KUKA KRL program: MyProgram_335().src

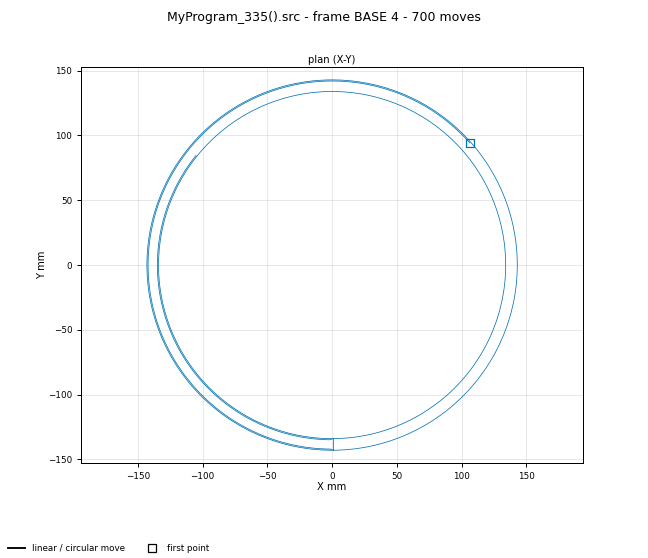
[picture p0: tool path of MyProgram_335().src in frame BASE 4, 700 of 700 moves have a stored position in this frame; points joined in program order, loops and branches not executed]
&ACCESS RVP
&REL 1
&PARAM TEMPLATE = C:\KRC\Roboter\Template\vorgabe
&PARAM EDITMASK = *
DEF MyProgram_335()
; ---- Setting reference (Base) ----
$BASE = BASE_DATA[4]

; --------------------------
; ---- Setting tool (TCP) ----
$TOOL = TOOL_DATA[3]
; --------------------------

$VEL.CP = VEL_APROX_PRINT
Startdeposition()
$VEL.CP = VEL_PRINT
LIN {X 106.2773,Y 94.2336,Z 189,A 42.7394,B 1.6929,C 0.0223,E1 1.815,E2 411.3828} C_DIS
LIN {X 103.2721,Y 97.5175,Z 189,A 44.3965,B 1.6929,C 0.0193,E1 1.8118,E2 409.7431} C_DIS
LIN {X 100.41,Y 100.4629,Z 189,A 45.7845,B 1.6929,C 0.0174,E1 1.8092,E2 408.3889} C_DIS
LIN {X 97.7243,Y 103.0771,Z 189,A 47.4179,B 1.693,C 0.0135,E1 1.8059,E2 406.7401} C_DIS
LIN {X 94.6798,Y 105.8799,Z 189,A 48.9807,B 1.693,C 0.0108,E1 1.8026,E2 405.1906} C_DIS
LIN {X 91.6362,Y 108.5256,Z 189,A 50.5192,B 1.693,C 0.0082,E1 1.7994,E2 403.6632} C_DIS
LIN {X 88.3912,Y 111.1836,Z 189,A 52.0959,B 1.693,C 0.0056,E1 1.796,E2 402.101} C_DIS
LIN {X 85.1125,Y 113.7136,Z 189,A 53.6495,B 1.693,C 0.0032,E1 1.7926,E2 400.562} C_DIS
LIN {X 81.9996,Y 115.978,Z 189,A 55.2099,B 1.693,C 0.0004,E1 1.789,E2 399.0007} C_DIS
LIN {X 78.1765,Y 118.5885,Z 189,A 56.9737,B 1.693,C -0.0023,E1 1.7849,E2 397.2499} C_DIS
LIN {X 74.3685,Y 121.013,Z 189,A 58.7195,B 1.693,C -0.0049,E1 1.7808,E2 395.5136} C_DIS
LIN {X 70.5126,Y 123.2996,Z 189,A 60.4494,B 1.693,C -0.0073,E1 1.7766,E2 393.7936} C_DIS
LIN {X 66.5595,Y 125.4767,Z 189,A 62.2164,B 1.693,C -0.0098,E1 1.7723,E2 392.0335} C_DIS
LIN {X 63.0559,Y 127.2723,Z 189,A 63.6578,B 1.693,C -0.0113,E1 1.7687,E2 390.6104} C_DIS
LIN {X 59.5637,Y 128.9434,Z 189,A 65.1264,B 1.693,C -0.013,E1 1.7651,E2 389.1536} C_DIS
LIN {X 56.8008,Y 130.185,Z 189,A 66.2211,B 1.693,C -0.014,E1 1.7623,E2 388.0748} C_DIS
LIN {X 54.0024,Y 131.372,Z 189,A 67.6332,B 1.693,C -0.0165,E1 1.7586,E2 386.64} C_DIS
LIN {X 50.101,Y 132.9068,Z 189,A 69.1211,B 1.693,C -0.0175,E1 1.7547,E2 385.1775} C_DIS
LIN {X 46.8537,Y 134.0862,Z 189,A 70.4786,B 1.693,C -0.019,E1 1.7512,E2 383.8248} C_DIS
LIN {X 40.2783,Y 136.206,Z 189,A 73.0708,B 1.693,C -0.021,E1 1.7443,E2 381.2572} C_DIS
LIN {X 36.9072,Y 137.1577,Z 189,A 74.5574,B 1.693,C -0.0227,E1 1.7403,E2 379.7619} C_DIS
LIN {X 33.8671,Y 137.9408,Z 189,A 75.7576,B 1.693,C -0.0236,E1 1.737,E2 378.5701} C_DIS
LIN {X 29.912,Y 138.8509,Z 189,A 77.2778,B 1.693,C -0.0244,E1 1.7329,E2 377.0648} C_DIS
LIN {X 27.0157,Y 139.4438,Z 189,A 78.5435,B 1.6929,C -0.0257,E1 1.7294,E2 375.7905} C_DIS
LIN {X 23.2743,Y 140.1165,Z 189,A 80.0251,B 1.6929,C -0.0266,E1 1.7253,E2 374.3156} C_DIS
LIN {X 19.566,Y 140.6833,Z 189,A 81.6158,B 1.6929,C -0.0279,E1 1.7209,E2 372.7159} C_DIS
LIN {X 15.4525,Y 141.1936,Z 189,A 83.1691,B 1.6929,C -0.0283,E1 1.7166,E2 371.1777} C_DIS
LIN {X 12.1084,Y 141.5195,Z 189,A 84.3357,B 1.6929,C -0.0283,E1 1.7134,E2 370.0346} C_DIS
LIN {X 9.4248,Y 141.7252,Z 189,A 85.5879,B 1.6929,C -0.0294,E1 1.7099,E2 368.7625} C_DIS
LIN {X 6.1391,Y 141.9051,Z 189,A 86.9513,B 1.6929,C -0.03,E1 1.706,E2 367.3953} C_DIS
LIN {X 1.6359,Y 142.029,Z 189,A 88.7776,B 1.6929,C -0.0306,E1 1.7009,E2 365.5686} C_DIS
LIN {X -2.4489,Y 142.0155,Z 189,A 90.3695,B 1.6929,C -0.0308,E1 1.6965,E2 363.9841} C_DIS
LIN {X -6.6903,Y 141.8796,Z 189,A 92.0648,B 1.6929,C -0.031,E1 1.6917,E2 362.2916} C_DIS
LIN {X -10.4141,Y 141.6542,Z 189,A 93.5286,B 1.6929,C -0.031,E1 1.6876,E2 360.8335} C_DIS
LIN {X -14.6574,Y 141.2792,Z 189,A 95.349,B 1.6928,C -0.0312,E1 1.6825,E2 359.0014} C_DIS
LIN {X -19.0699,Y 140.7518,Z 189,A 97.1416,B 1.6928,C -0.0311,E1 1.6775,E2 357.2096} C_DIS
LIN {X -22.6456,Y 140.2214,Z 189,A 98.4481,B 1.6928,C -0.0303,E1 1.674,E2 355.9224} C_DIS
LIN {X -26.2848,Y 139.5836,Z 189,A 99.9509,B 1.6928,C -0.0299,E1 1.6698,E2 354.4187} C_DIS
LIN {X -30.2845,Y 138.7705,Z 189,A 101.8492,B 1.6928,C -0.0302,E1 1.6645,E2 352.4905} C_DIS
LIN {X -34.665,Y 137.7415,Z 189,A 103.4007,B 1.6928,C -0.0286,E1 1.6604,E2 350.9722} C_DIS
LIN {X -38.3306,Y 136.7664,Z 189,A 105.04,B 1.6928,C -0.0282,E1 1.6559,E2 349.3203} C_DIS
LIN {X -41.5195,Y 135.8322,Z 189,A 106.3705,B 1.6928,C -0.0274,E1 1.6523,E2 347.9917} C_DIS
LIN {X -44.6408,Y 134.8389,Z 189,A 107.699,B 1.6928,C -0.0266,E1 1.6488,E2 346.6631} C_DIS
LIN {X -47.2057,Y 133.9641,Z 189,A 109.0092,B 1.6928,C -0.0264,E1 1.6453,E2 345.3271} C_DIS
LIN {X -51.3738,Y 132.4197,Z 189,A 110.6484,B 1.6929,C -0.0247,E1 1.641,E2 343.7076} C_DIS
LIN {X -53.9048,Y 131.4126,Z 189,A 111.9788,B 1.6929,C -0.0244,E1 1.6375,E2 342.3496} C_DIS
LIN {X -57.1041,Y 130.0538,Z 189,A 113.2798,B 1.6929,C -0.0228,E1 1.6342,E2 341.0619} C_DIS
LIN {X -60.454,Y 128.5312,Z 189,A 115.0186,B 1.6929,C -0.022,E1 1.6297,E2 339.2927} C_DIS
LIN {X -64.3455,Y 126.6249,Z 189,A 116.6404,B 1.6929,C -0.0199,E1 1.6257,E2 337.6873} C_DIS
LIN {X -67.2006,Y 125.1355,Z 189,A 118.1653,B 1.6929,C -0.019,E1 1.6218,E2 336.1356} C_DIS
LIN {X -71.656,Y 122.639,Z 189,A 120.235,B 1.693,C -0.0166,E1 1.6168,E2 334.066} C_DIS
LIN {X -75.5784,Y 120.2613,Z 189,A 122.1545,B 1.693,C -0.0143,E1 1.6122,E2 332.1392} C_DIS
LIN {X -79.4708,Y 117.7252,Z 189,A 124.0179,B 1.693,C -0.0118,E1 1.6078,E2 330.2783} C_DIS
LIN {X -83.1126,Y 115.1833,Z 189,A 125.9602,B 1.693,C -0.0095,E1 1.6034,E2 328.3184} C_DIS
LIN {X -86.7314,Y 112.4837,Z 189,A 127.8838,B 1.693,C -0.0069,E1 1.599,E2 326.3833} C_DIS
LIN {X -90.284,Y 109.6528,Z 189,A 129.7857,B 1.693,C -0.0041,E1 1.5949,E2 324.4741} C_DIS
LIN {X -93.551,Y 106.8787,Z 189,A 131.6035,B 1.693,C -0.0013,E1 1.591,E2 322.6463} C_DIS
LIN {X -96.9568,Y 103.799,Z 189,A 133.5203,B 1.693,C 0.0018,E1 1.5871,E2 320.7227} C_DIS
LIN {X -100.085,Y 100.7858,Z 189,A 135.4048,B 1.693,C 0.0048,E1 1.5833,E2 318.823} C_DIS
LIN {X -103.2004,Y 97.5936,Z 189,A 137.3305,B 1.693,C 0.008,E1 1.5795,E2 316.8826} C_DIS
LIN {X -106.2595,Y 94.2537,Z 189,A 139.2838,B 1.693,C 0.0114,E1 1.5758,E2 314.9147} C_DIS
LIN {X -109.2471,Y 90.774,Z 189,A 141.2114,B 1.693,C 0.0151,E1 1.5723,E2 312.9787} C_DIS
LIN {X -111.9901,Y 87.3683,Z 189,A 142.9572,B 1.693,C 0.0188,E1 1.5693,E2 311.2364} C_DIS
LIN {X -114.18,Y 84.4857,Z 189,A 144.7828,B 1.693,C 0.0214,E1 1.5661,E2 309.3657} C_DIS
LIN {X -117.2007,Y 80.2423,Z 189,A 146.9388,B 1.6929,C 0.026,E1 1.5627,E2 307.2043} C_DIS
LIN {X -119.775,Y 76.3468,Z 189,A 148.9107,B 1.6929,C 0.0302,E1 1.5597,E2 305.2224} C_DIS
LIN {X -122.0067,Y 72.7266,Z 189,A 150.7317,B 1.6927,C 0.0341,E1 1.557,E2 303.3893} C_DIS
LIN {X -124.3948,Y 68.5625,Z 189,A 152.8841,B 1.6927,C 0.0384,E1 1.554,E2 301.2106} C_DIS
LIN {X -126.4099,Y 64.7679,Z 189,A 154.6626,B 1.6925,C 0.0426,E1 1.5517,E2 299.4275} C_DIS
LIN {X -129.3506,Y 58.6788,Z 189,A 157.6639,B 1.6924,C 0.0491,E1 1.5481,E2 296.3931} C_DIS
LIN {X -131.2019,Y 54.4098,Z 189,A 159.744,B 1.6922,C 0.0537,E1 1.5458,E2 294.2881} C_DIS
LIN {X -132.6655,Y 50.7415,Z 189,A 161.5557,B 1.6922,C 0.0576,E1 1.5439,E2 292.4493} C_DIS
LIN {X -133.971,Y 47.1847,Z 189,A 162.9511,B 1.692,C 0.0617,E1 1.5426,E2 291.0722} C_DIS
LIN {X -135.1927,Y 43.5582,Z 189,A 164.6541,B 1.6918,C 0.0656,E1 1.5411,E2 289.3496} C_DIS
LIN {X -136.1268,Y 40.5488,Z 189,A 166.2155,B 1.6917,C 0.0688,E1 1.5398,E2 287.7514} C_DIS
LIN {X -138.2076,Y 32.7602,Z 189,A 169.5503,B 1.6913,C 0.0775,E1 1.5375,E2 284.408} C_DIS
LIN {X -139.5086,Y 26.6769,Z 189,A 172.3268,B 1.691,C 0.0842,E1 1.5359,E2 281.5983} C_DIS
LIN {X -140.4655,Y 21.0763,Z 189,A 174.9757,B 1.6907,C 0.0902,E1 1.5346,E2 278.9039} C_DIS
LIN {X -141.0217,Y 16.9484,Z 189,A 176.6676,B 1.6904,C 0.0949,E1 1.534,E2 277.2115} C_DIS
LIN {X -141.332,Y 14.1401,Z 189,A 177.8354,B 1.6902,C 0.098,E1 1.5337,E2 276.0408} C_DIS
LIN {X -141.6373,Y 10.6462,Z 189,A 179.4383,B 1.69,C 0.1018,E1 1.5333,E2 274.4138} C_DIS
LIN {X -141.8039,Y 8.1466,Z 189,A -179.2535,B 1.6899,C 0.1044,E1 1.5331,E2 273.0667} C_DIS
LIN {X -141.9587,Y 4.7647,Z 189,A -177.7459,B 1.6896,C 0.1081,E1 1.533,E2 271.5411} C_DIS
LIN {X -142.0388,Y -0.2591,Z 189,A -175.4645,B 1.6893,C 0.1136,E1 1.533,E2 269.2268} C_DIS
LIN {X -141.9528,Y -4.9149,Z 189,A -173.7364,B 1.6889,C 0.119,E1 1.533,E2 267.5199} C_DIS
LIN {X -141.8556,Y -7.1668,Z 189,A -172.5939,B 1.6887,C 0.1213,E1 1.5332,E2 266.3465} C_DIS
LIN {X -141.4766,Y -12.6168,Z 189,A -170.148,B 1.6883,C 0.1273,E1 1.5337,E2 263.8692} C_DIS
LIN {X -141.0326,Y -16.8571,Z 189,A -168.4784,B 1.6879,C 0.1321,E1 1.5342,E2 262.2073} C_DIS
LIN {X -140.629,Y -19.9456,Z 189,A -166.1435,B 1.6877,C 0.1346,E1 1.5353,E2 259.7262} C_DIS
LIN {X -139.6388,Y -25.996,Z 189,A -163.7081,B 1.6872,C 0.1414,E1 1.5365,E2 257.2973} C_DIS
LIN {X -138.6976,Y -30.6224,Z 189,A -162.0866,B 1.6867,C 0.1469,E1 1.5374,E2 255.7156} C_DIS
LIN {X -137.8516,Y -34.231,Z 189,A -160.4161,B 1.6864,C 0.1507,E1 1.5385,E2 254.0218} C_DIS
LIN {X -136.7518,Y -38.3827,Z 189,A -158.7867,B 1.6859,C 0.1555,E1 1.5397,E2 252.4073} C_DIS
LIN {X -135.9501,Y -41.1344,Z 189,A -157.4275,B 1.6857,C 0.1583,E1 1.5408,E2 251.0207} C_DIS
LIN {X -135.008,Y -44.133,Z 189,A -155.8637,B 1.6854,C 0.1613,E1 1.5422,E2 249.4167} C_DIS
LIN {X -133.8121,Y -47.6331,Z 189,A -154.5652,B 1.685,C 0.1654,E1 1.5434,E2 248.1456} C_DIS
LIN {X -132.7591,Y -50.4955,Z 189,A -152.9409,B 1.6847,C 0.1682,E1 1.545,E2 246.4674} C_DIS
LIN {X -131.2624,Y -54.2648,Z 189,A -151.4833,B 1.6843,C 0.1725,E1 1.5465,E2 245.035} C_DIS
LIN {X -128.9947,Y -59.4527,Z 189,A -148.7099,B 1.6837,C 0.1776,E1 1.5497,E2 242.1946} C_DIS
LIN {X -126.7671,Y -64.0663,Z 189,A -146.6066,B 1.6832,C 0.1826,E1 1.5523,E2 240.0869} C_DIS
LIN {X -125.0385,Y -67.3811,Z 189,A -144.9402,B 1.6828,C 0.186,E1 1.5546,E2 238.399} C_DIS
LIN {X -122.8547,Y -71.2849,Z 189,A -143.0116,B 1.6824,C 0.1901,E1 1.5572,E2 236.4535} C_DIS
LIN {X -121.0931,Y -74.2378,Z 189,A -141.2058,B 1.6821,C 0.1926,E1 1.56,E2 234.5893} C_DIS
LIN {X -119.1112,Y -77.3777,Z 189,A -140.0244,B 1.6816,C 0.1965,E1 1.5617,E2 233.4528} C_DIS
LIN {X -116.9843,Y -80.5575,Z 189,A -138.2365,B 1.6813,C 0.1995,E1 1.5645,E2 231.6308} C_DIS
LIN {X -115.1472,Y -83.1624,Z 189,A -136.5306,B 1.681,C 0.2016,E1 1.5675,E2 229.8659} C_DIS
LIN {X -112.8126,Y -86.3024,Z 189,A -135.1781,B 1.6806,C 0.2053,E1 1.5697,E2 228.5457} C_DIS
LIN {X -110.1042,Y -89.7324,Z 189,A -133.3246,B 1.6802,C 0.2088,E1 1.5729,E2 226.6797} C_DIS
LIN {X -108.1098,Y -92.1254,Z 189,A -131.8953,B 1.6799,C 0.211,E1 1.5756,E2 225.2261} C_DIS
LIN {X -104.9235,Y -95.7393,Z 189,A -129.8541,B 1.6794,C 0.2145,E1 1.5794,E2 223.1713} C_DIS
LIN {X -101.7136,Y -99.143,Z 189,A -127.698,B 1.6791,C 0.2175,E1 1.5837,E2 220.9771} C_DIS
LIN {X -98.0261,Y -102.7896,Z 189,A -125.6758,B 1.6786,C 0.2214,E1 1.5877,E2 218.965} C_DIS
LIN {X -94.5718,Y -105.9766,Z 189,A -123.6873,B 1.6781,C 0.2244,E1 1.5919,E2 216.9634} C_DIS
LIN {X -91.0557,Y -109.0126,Z 189,A -121.6766,B 1.6778,C 0.2271,E1 1.5962,E2 214.9332} C_DIS
LIN {X -87.3782,Y -111.9823,Z 189,A -119.7857,B 1.6774,C 0.2301,E1 1.6003,E2 213.0446} C_DIS
LIN {X -83.6065,Y -114.8253,Z 189,A -117.6892,B 1.6771,C 0.2325,E1 1.6051,E2 210.9206} C_DIS
LIN {X -79.8824,Y -117.4466,Z 189,A -115.7606,B 1.6767,C 0.2348,E1 1.6096,E2 208.9788} C_DIS
LIN {X -75.983,Y -120.0059,Z 189,A -113.8584,B 1.6764,C 0.2372,E1 1.6141,E2 207.0734} C_DIS
LIN {X -72.2327,Y -122.3002,Z 189,A -111.9585,B 1.6761,C 0.239,E1 1.6187,E2 205.1552} C_DIS
LIN {X -68.162,Y -124.6145,Z 189,A -110.0444,B 1.6758,C 0.241,E1 1.6234,E2 203.2372} C_DIS
LIN {X -64.7484,Y -126.4198,Z 189,A -108.5031,B 1.6756,C 0.2427,E1 1.6272,E2 201.698} C_DIS
LIN {X -61.576,Y -127.9952,Z 189,A -107.1255,B 1.6754,C 0.2443,E1 1.6307,E2 200.3275} C_DIS
LIN {X -58.3162,Y -129.5128,Z 189,A -105.7448,B 1.6751,C 0.2459,E1 1.6342,E2 198.9566} C_DIS
LIN {X -55.7418,Y -130.6428,Z 189,A -104.2642,B 1.6751,C 0.2457,E1 1.6381,E2 197.4258} C_DIS
LIN {X -51.8273,Y -132.2434,Z 189,A -102.6432,B 1.6749,C 0.2473,E1 1.6423,E2 195.8167} C_DIS
LIN {X -48.4711,Y -133.5099,Z 189,A -101.2597,B 1.6747,C 0.2486,E1 1.6459,E2 194.442} C_DIS
LIN {X -43.7182,Y -135.1416,Z 189,A -98.9872,B 1.6747,C 0.249,E1 1.652,E2 192.1334} C_DIS
LIN {X -39.1432,Y -136.5384,Z 189,A -97.0299,B 1.6745,C 0.2499,E1 1.6573,E2 190.1717} C_DIS
LIN {X -34.3439,Y -137.8229,Z 189,A -94.9798,B 1.6745,C 0.2506,E1 1.6629,E2 188.1142} C_DIS
LIN {X -30.6716,Y -138.6869,Z 189,A -93.6287,B 1.6743,C 0.2518,E1 1.6665,E2 186.7874} C_DIS
LIN {X -27.0587,Y -139.4356,Z 189,A -91.9873,B 1.6743,C 0.2516,E1 1.6711,E2 185.1231} C_DIS
LIN {X -23.8319,Y -140.0235,Z 189,A -90.8191,B 1.6742,C 0.2525,E1 1.6743,E2 183.9769} C_DIS
LIN {X -20.9337,Y -140.4876,Z 189,A -89.3995,B 1.6742,C 0.2517,E1 1.6783,E2 182.5227} C_DIS
LIN {X -16.9659,Y -141.0196,Z 189,A -88.0583,B 1.6741,C 0.253,E1 1.6819,E2 181.2205} C_DIS
LIN {X -14.208,Y -141.3255,Z 189,A -86.8707,B 1.6741,C 0.2527,E1 1.6853,E2 180.0226} C_DIS
LIN {X -10.3399,Y -141.6596,Z 189,A -85.1907,B 1.6742,C 0.2521,E1 1.69,E2 178.3253} C_DIS
LIN {X -5.7286,Y -141.9211,Z 189,A -83.3211,B 1.6742,C 0.2519,E1 1.6953,E2 176.4539} C_DIS
LIN {X -1.1428,Y -142.0324,Z 189,A -81.5425,B 1.6742,C 0.2518,E1 1.7002,E2 174.6848} C_DIS
LIN {X -1.1428,Y -142.0324,Z 189,A -81.5425,B 1.6742,C 0.2518,E1 1.7002,E2 174.6848} C_DIS
Enddeposition()
LIN {X 1.0097,Y -142.9296,Z 189,A -80.9147,B 1.6738,C 0.2534,E1 1.7016,E2 174.1194} C_DIS
Startdeposition()
$VEL.CP = VEL_PRINT
LIN {X -1.408,Y -142.9302,Z 189,A -82.2099,B 1.6736,C 0.2552,E1 1.6979,E2 175.4628} C_DIS
LIN {X -5.2622,Y -142.8391,Z 189,A -83.6981,B 1.6736,C 0.2552,E1 1.6937,E2 176.9434} C_DIS
LIN {X -8.4198,Y -142.6879,Z 189,A -85.1105,B 1.6734,C 0.256,E1 1.6897,E2 178.3774} C_DIS
LIN {X -12.2561,Y -142.4094,Z 189,A -86.5262,B 1.6735,C 0.2555,E1 1.6858,E2 179.7755} C_DIS
LIN {X -15.4038,Y -142.1032,Z 189,A -87.8442,B 1.6735,C 0.2557,E1 1.6821,E2 181.1013} C_DIS
LIN {X -19.2397,Y -141.6364,Z 189,A -89.3872,B 1.6735,C 0.2557,E1 1.6778,E2 182.6442} C_DIS
LIN {X -22.7055,Y -141.123,Z 189,A -90.8211,B 1.6735,C 0.2555,E1 1.6738,E2 184.083} C_DIS
LIN {X -25.7283,Y -140.602,Z 189,A -92.0459,B 1.6735,C 0.2552,E1 1.6704,E2 185.3074} C_DIS
LIN {X -29.4561,Y -139.8692,Z 189,A -93.6335,B 1.6735,C 0.255,E1 1.666,E2 186.905} C_DIS
LIN {X -33.0187,Y -139.0702,Z 189,A -95.0391,B 1.6737,C 0.2543,E1 1.6622,E2 188.3027} C_DIS
LIN {X -36.4297,Y -138.2157,Z 189,A -96.3842,B 1.6738,C 0.2535,E1 1.6586,E2 189.6389} C_DIS
LIN {X -39.7974,Y -137.2837,Z 189,A -97.8075,B 1.6739,C 0.2529,E1 1.6547,E2 191.066} C_DIS
LIN {X -42.824,Y -136.3712,Z 189,A -99.198,B 1.6739,C 0.2526,E1 1.6509,E2 192.4747} C_DIS
LIN {X -46.4642,Y -135.1729,Z 189,A -100.6617,B 1.6741,C 0.2514,E1 1.6471,E2 193.9283} C_DIS
LIN {X -49.0106,Y -134.2712,Z 189,A -102.0278,B 1.6741,C 0.2516,E1 1.6434,E2 195.3356} C_DIS
LIN {X -53.0801,Y -132.7144,Z 189,A -103.5446,B 1.6744,C 0.2495,E1 1.6395,E2 196.8196} C_DIS
LIN {X -56.0011,Y -131.5103,Z 189,A -104.9545,B 1.6745,C 0.2489,E1 1.6358,E2 198.2506} C_DIS
LIN {X -58.7218,Y -130.3164,Z 189,A -106.1866,B 1.6746,C 0.248,E1 1.6326,E2 199.4888} C_DIS
LIN {X -61.8977,Y -128.838,Z 189,A -107.6334,B 1.6748,C 0.2468,E1 1.6289,E2 200.942} C_DIS
LIN {X -65.0427,Y -127.279,Z 189,A -109.0825,B 1.675,C 0.2455,E1 1.6253,E2 202.3974} C_DIS
LIN {X -68.3071,Y -125.5595,Z 189,A -110.7111,B 1.6752,C 0.2443,E1 1.6212,E2 204.0477} C_DIS
LIN {X -71.9805,Y -123.491,Z 189,A -112.3949,B 1.6755,C 0.2423,E1 1.6171,E2 205.7309} C_DIS
LIN {X -75.5848,Y -121.3177,Z 189,A -114.1419,B 1.6757,C 0.2404,E1 1.6129,E2 207.4866} C_DIS
LIN {X -79.2667,Y -118.9447,Z 189,A -115.9737,B 1.676,C 0.2383,E1 1.6086,E2 209.3295} C_DIS
LIN {X -82.4457,Y -116.7637,Z 189,A -117.6742,B 1.6763,C 0.2366,E1 1.6046,E2 211.0522} C_DIS
LIN {X -85.9738,Y -114.1909,Z 189,A -119.4814,B 1.6766,C 0.2341,E1 1.6006,E2 212.8677} C_DIS
LIN {X -89.4478,Y -111.4911,Z 189,A -121.3704,B 1.677,C 0.2317,E1 1.5964,E2 214.7746} C_DIS
LIN {X -92.704,Y -108.7981,Z 189,A -123.1445,B 1.6773,C 0.2292,E1 1.5925,E2 216.56} C_DIS
LIN {X -96.115,Y -105.7967,Z 189,A -125.0599,B 1.6777,C 0.2263,E1 1.5885,E2 218.4887} C_DIS
LIN {X -99.3067,Y -102.8068,Z 189,A -126.8794,B 1.6781,C 0.2233,E1 1.5848,E2 220.3175} C_DIS
LIN {X -102.2872,Y -99.8423,Z 189,A -128.5767,B 1.6785,C 0.2203,E1 1.5815,E2 222.0164} C_DIS
LIN {X -105.2002,Y -96.7675,Z 189,A -130.4002,B 1.6789,C 0.2173,E1 1.5779,E2 223.8574} C_DIS
LIN {X -108.0446,Y -93.5818,Z 189,A -132.2121,B 1.6793,C 0.2142,E1 1.5746,E2 225.6833} C_DIS
LIN {X -110.4898,Y -90.6814,Z 189,A -133.9376,B 1.6796,C 0.2115,E1 1.5714,E2 227.4374} C_DIS
LIN {X -113.2109,Y -87.261,Z 189,A -135.7018,B 1.6801,C 0.2078,E1 1.5684,E2 229.203} C_DIS
LIN {X -115.7265,Y -83.8952,Z 189,A -137.5131,B 1.6805,C 0.2045,E1 1.5653,E2 231.0318} C_DIS
LIN {X -118.2614,Y -80.2827,Z 189,A -139.3933,B 1.681,C 0.2008,E1 1.5623,E2 232.9272} C_DIS
LIN {X -120.365,Y -77.0927,Z 189,A -141.1327,B 1.6813,C 0.1976,E1 1.5596,E2 234.6953} C_DIS
LIN {X -122.6017,Y -73.4845,Z 189,A -142.9789,B 1.6818,C 0.1939,E1 1.5569,E2 236.5612} C_DIS
LIN {X -124.8787,Y -69.5448,Z 189,A -144.9149,B 1.6822,C 0.1898,E1 1.5542,E2 238.5123} C_DIS
LIN {X -126.7901,Y -65.9924,Z 189,A -146.5547,B 1.6827,C 0.186,E1 1.5521,E2 240.1547} C_DIS
LIN {X -128.3777,Y -62.8474,Z 189,A -148.0738,B 1.683,C 0.1827,E1 1.5502,E2 241.6881} C_DIS
LIN {X -129.8804,Y -59.6797,Z 189,A -149.5912,B 1.6834,C 0.1793,E1 1.5483,E2 243.2205} C_DIS
LIN {X -131.3588,Y -56.3515,Z 189,A -151.1443,B 1.6838,C 0.1758,E1 1.5466,E2 244.786} C_DIS
LIN {X -132.7165,Y -53.0751,Z 189,A -152.664,B 1.6841,C 0.1723,E1 1.545,E2 246.3187} C_DIS
LIN {X -133.8564,Y -50.1293,Z 189,A -154.1378,B 1.6844,C 0.1693,E1 1.5435,E2 247.8206} C_DIS
LIN {X -135.1558,Y -46.5134,Z 189,A -155.7021,B 1.6848,C 0.1653,E1 1.542,E2 249.3876} C_DIS
LIN {X -136.158,Y -43.4913,Z 189,A -157.1951,B 1.6851,C 0.1622,E1 1.5407,E2 250.9097} C_DIS
LIN {X -137.2796,Y -39.8117,Z 189,A -158.7686,B 1.6855,C 0.1581,E1 1.5395,E2 252.4869} C_DIS
LIN {X -138.1263,Y -36.7647,Z 189,A -160.1953,B 1.6858,C 0.1549,E1 1.5384,E2 253.9348} C_DIS
LIN {X -138.9874,Y -33.3623,Z 189,A -161.7271,B 1.6861,C 0.1512,E1 1.5374,E2 255.4829} C_DIS
LIN {X -139.7645,Y -29.941,Z 189,A -163.2595,B 1.6865,C 0.1475,E1 1.5364,E2 257.0318} C_DIS
LIN {X -140.5199,Y -26.1755,Z 189,A -164.912,B 1.6868,C 0.1434,E1 1.5355,E2 258.6989} C_DIS
LIN {X -141.0622,Y -23.0699,Z 189,A -166.3064,B 1.6871,C 0.1401,E1 1.5349,E2 260.1104} C_DIS
LIN {X -141.5904,Y -19.5744,Z 189,A -167.8479,B 1.6874,C 0.1363,E1 1.5342,E2 261.668} C_DIS
LIN {X -142.0642,Y -15.7664,Z 189,A -169.5501,B 1.6877,C 0.1321,E1 1.5337,E2 263.3914} C_DIS
LIN {X -142.4066,Y -12.2889,Z 189,A -170.9826,B 1.688,C 0.1282,E1 1.5333,E2 264.8274} C_DIS
LIN {X -142.6438,Y -9.1356,Z 189,A -172.5371,B 1.6883,C 0.1249,E1 1.533,E2 266.4197} C_DIS
LIN {X -142.8393,Y -5.2579,Z 189,A -174.0995,B 1.6886,C 0.1206,E1 1.5328,E2 267.982} C_DIS
LIN {X -142.9205,Y -2.1023,Z 189,A -175.517,B 1.6888,C 0.1172,E1 1.5328,E2 269.4191} C_DIS
LIN {X -142.9314,Y 1.2571,Z 189,A -177.1181,B 1.6891,C 0.1136,E1 1.5328,E2 271.0533} C_DIS
LIN {X -142.8394,Y 5.2564,Z 189,A -178.6726,B 1.6894,C 0.1091,E1 1.5328,E2 272.6004} C_DIS
LIN {X -142.6874,Y 8.4286,Z 189,A 179.7693,B 1.6896,C 0.1057,E1 1.5331,E2 274.1955} C_DIS
LIN {X -142.4177,Y 12.1579,Z 189,A 178.2546,B 1.6899,C 0.1016,E1 1.5334,E2 275.7114} C_DIS
LIN {X -142.1033,Y 15.4032,Z 189,A 176.7863,B 1.6901,C 0.098,E1 1.5339,E2 277.2001} C_DIS
LIN {X -141.6393,Y 19.2174,Z 189,A 175.1147,B 1.6903,C 0.0939,E1 1.5345,E2 278.8881} C_DIS
LIN {X -141.1264,Y 22.6839,Z 189,A 173.5843,B 1.6905,C 0.0901,E1 1.5351,E2 280.4341} C_DIS
LIN {X -140.6101,Y 25.6829,Z 189,A 172.2359,B 1.6907,C 0.0868,E1 1.5358,E2 281.7985} C_DIS
LIN {X -139.8447,Y 29.5695,Z 189,A 170.5028,B 1.6909,C 0.0826,E1 1.5367,E2 283.5496} C_DIS
LIN {X -139.082,Y 32.97,Z 189,A 168.9809,B 1.6911,C 0.0789,E1 1.5377,E2 285.0868} C_DIS
LIN {X -138.1442,Y 36.6977,Z 189,A 167.2273,B 1.6912,C 0.0749,E1 1.539,E2 286.867} C_DIS
LIN {X -136.8823,Y 41.1612,Z 189,A 165.2802,B 1.6915,C 0.07,E1 1.5405,E2 288.8243} C_DIS
LIN {X -135.7167,Y 44.8505,Z 189,A 163.5964,B 1.6916,C 0.066,E1 1.5419,E2 290.5241} C_DIS
LIN {X -134.6949,Y 47.8354,Z 189,A 162.2243,B 1.6917,C 0.0628,E1 1.5432,E2 291.9093} C_DIS
LIN {X -133.455,Y 51.1924,Z 189,A 160.5899,B 1.6919,C 0.0592,E1 1.5448,E2 293.5684} C_DIS
LIN {X -132.1903,Y 54.3763,Z 189,A 159.1817,B 1.6919,C 0.0557,E1 1.5463,E2 294.9801} C_DIS
LIN {X -130.8136,Y 57.6102,Z 189,A 157.6716,B 1.6921,C 0.0523,E1 1.548,E2 296.5022} C_DIS
LIN {X -129.5944,Y 60.2982,Z 189,A 156.3682,B 1.6921,C 0.0494,E1 1.5496,E2 297.8201} C_DIS
LIN {X -127.7947,Y 64.0292,Z 189,A 154.5685,B 1.6923,C 0.0455,E1 1.5518,E2 299.6366} C_DIS
LIN {X -126.1391,Y 67.2322,Z 189,A 153.0106,B 1.6923,C 0.0421,E1 1.5538,E2 301.2078} C_DIS
LIN {X -124.3581,Y 70.4717,Z 189,A 151.4211,B 1.6925,C 0.0387,E1 1.556,E2 302.8098} C_DIS
LIN {X -122.5083,Y 73.6403,Z 189,A 149.7209,B 1.6925,C 0.0355,E1 1.5585,E2 304.538} C_DIS
LIN {X -120.2912,Y 77.2081,Z 189,A 147.8888,B 1.6926,C 0.0318,E1 1.5612,E2 306.3876} C_DIS
LIN {X -117.7768,Y 80.9919,Z 189,A 145.9368,B 1.6926,C 0.0278,E1 1.5643,E2 308.3548} C_DIS
LIN {X -114.9265,Y 84.989,Z 189,A 143.8604,B 1.6927,C 0.0237,E1 1.5677,E2 310.4434} C_DIS
LIN {X -112.143,Y 88.6294,Z 189,A 141.9924,B 1.6927,C 0.0198,E1 1.571,E2 312.3141} C_DIS
LIN {X -109.8275,Y 91.4829,Z 189,A 140.2818,B 1.6928,C 0.0171,E1 1.5741,E2 314.0533} C_DIS
LIN {X -106.6192,Y 95.202,Z 189,A 138.2635,B 1.6928,C 0.0133,E1 1.5778,E2 316.0764} C_DIS
LIN {X -103.5205,Y 98.5628,Z 189,A 136.3937,B 1.6928,C 0.0098,E1 1.5814,E2 317.9495} C_DIS
LIN {X -101.0738,Y 101.0709,Z 189,A 134.7774,B 1.6928,C 0.0075,E1 1.5846,E2 319.5912} C_DIS
LIN {X -97.9296,Y 104.1195,Z 189,A 132.9049,B 1.6928,C 0.0046,E1 1.5884,E2 321.477} C_DIS
LIN {X -94.5507,Y 107.1971,Z 189,A 130.9743,B 1.6928,C 0.0016,E1 1.5925,E2 323.4185} C_DIS
LIN {X -90.8118,Y 110.3832,Z 189,A 128.9328,B 1.6928,C -0.0015,E1 1.5969,E2 325.4676} C_DIS
LIN {X -87.2518,Y 113.218,Z 189,A 127.0909,B 1.6928,C -0.0044,E1 1.6009,E2 327.3105} C_DIS
LIN {X -83.8809,Y 115.7369,Z 189,A 125.3172,B 1.6928,C -0.0067,E1 1.6049,E2 329.0937} C_DIS
LIN {X -80.279,Y 118.2639,Z 189,A 123.4755,B 1.6928,C -0.009,E1 1.6092,E2 330.9439} C_DIS
LIN {X -77.0705,Y 120.3793,Z 189,A 121.7791,B 1.6928,C -0.0108,E1 1.6132,E2 332.6583} C_DIS
LIN {X -72.8912,Y 122.9554,Z 189,A 119.8529,B 1.6928,C -0.0134,E1 1.6178,E2 334.5782} C_DIS
LIN {X -69.5572,Y 124.8718,Z 189,A 118.15,B 1.6928,C -0.0148,E1 1.622,E2 336.2999} C_DIS
LIN {X -65.9644,Y 126.8048,Z 189,A 116.5603,B 1.6928,C -0.0167,E1 1.626,E2 337.883} C_DIS
LIN {X -63.036,Y 128.2847,Z 189,A 115.2099,B 1.6928,C -0.018,E1 1.6294,E2 339.2368} C_DIS
LIN {X -59.6042,Y 129.9153,Z 189,A 113.6446,B 1.6928,C -0.0194,E1 1.6333,E2 340.8063} C_DIS
LIN {X -56.0088,Y 131.507,Z 189,A 111.8888,B 1.6928,C -0.0203,E1 1.6379,E2 342.5831} C_DIS
LIN {X -51.7638,Y 133.2328,Z 189,A 110.0829,B 1.6928,C -0.0219,E1 1.6426,E2 344.3841} C_DIS
LIN {X -48.1615,Y 134.5774,Z 189,A 108.5583,B 1.6928,C -0.0231,E1 1.6466,E2 345.9059} C_DIS
LIN {X -45.1729,Y 135.6094,Z 189,A 107.2122,B 1.6928,C -0.0237,E1 1.6502,E2 347.2609} C_DIS
LIN {X -40.7977,Y 136.9908,Z 189,A 105.2315,B 1.6928,C -0.0244,E1 1.6556,E2 349.2577} C_DIS
LIN {X -36.7448,Y 138.1316,Z 189,A 103.6334,B 1.6928,C -0.0255,E1 1.6599,E2 350.844} C_DIS
LIN {X -33.0322,Y 139.067,Z 189,A 102.0438,B 1.6928,C -0.026,E1 1.6642,E2 352.4395} C_DIS
LIN {X -28.2201,Y 140.1223,Z 189,A 100.1003,B 1.6927,C -0.0267,E1 1.6695,E2 354.3782} C_DIS
LIN {X -24.7801,Y 140.7717,Z 189,A 98.7206,B 1.6927,C -0.0272,E1 1.6733,E2 355.7543} C_DIS
LIN {X -21.3239,Y 141.337,Z 189,A 97.3126,B 1.6927,C -0.0274,E1 1.6772,E2 357.1622} C_DIS
LIN {X -17.8526,Y 141.8181,Z 189,A 95.808,B 1.6927,C -0.0272,E1 1.6814,E2 358.6783} C_DIS
LIN {X -14.4077,Y 142.2096,Z 189,A 94.3868,B 1.6927,C -0.0272,E1 1.6854,E2 360.1027} C_DIS
LIN {X -10.8595,Y 142.5232,Z 189,A 93.0636,B 1.6927,C -0.0275,E1 1.6891,E2 361.4125} C_DIS
LIN {X -7.022,Y 142.7632,Z 189,A 91.6202,B 1.6927,C -0.0277,E1 1.6931,E2 362.8433} C_DIS
LIN {X -3.8617,Y 142.8836,Z 189,A 90.2801,B 1.6927,C -0.0273,E1 1.6969,E2 364.1917} C_DIS
LIN {X -0.0053,Y 142.9379,Z 189,A 88.7711,B 1.6927,C -0.0271,E1 1.7011,E2 365.6957} C_DIS
LIN {X 3.5072,Y 142.8934,Z 189,A 87.3317,B 1.6927,C -0.0265,E1 1.7051,E2 367.1383} C_DIS
LIN {X 6.6668,Y 142.781,Z 189,A 86.0778,B 1.6927,C -0.0261,E1 1.7086,E2 368.3901} C_DIS
LIN {X 10.5043,Y 142.5492,Z 189,A 84.5727,B 1.6927,C -0.0256,E1 1.7128,E2 369.8903} C_DIS
LIN {X 13.6556,Y 142.2818,Z 189,A 83.3209,B 1.6927,C -0.025,E1 1.7163,E2 371.1396} C_DIS
LIN {X 17.1578,Y 141.9022,Z 189,A 81.9044,B 1.6927,C -0.0242,E1 1.7203,E2 372.5562} C_DIS
LIN {X 20.9696,Y 141.391,Z 189,A 80.4392,B 1.6927,C -0.0235,E1 1.7243,E2 374.0117} C_DIS
LIN {X 24.4284,Y 140.8346,Z 189,A 79.0342,B 1.6927,C -0.0225,E1 1.7282,E2 375.4164} C_DIS
LIN {X 27.5463,Y 140.2578,Z 189,A 77.7267,B 1.6927,C -0.0214,E1 1.7318,E2 376.7279} C_DIS
LIN {X 31.3059,Y 139.466,Z 189,A 76.2899,B 1.6927,C -0.0206,E1 1.7357,E2 378.1516} C_DIS
LIN {X 34.6176,Y 138.6811,Z 189,A 74.9392,B 1.6927,C -0.0194,E1 1.7394,E2 379.5003} C_DIS
LIN {X 38.1028,Y 137.7638,Z 189,A 73.5655,B 1.6927,C -0.0184,E1 1.7431,E2 380.865} C_DIS
LIN {X 41.46,Y 136.7908,Z 189,A 72.1348,B 1.6928,C -0.0168,E1 1.7469,E2 382.299} C_DIS
LIN {X 45.6719,Y 135.4432,Z 189,A 70.4133,B 1.6928,C -0.0151,E1 1.7515,E2 384.0139} C_DIS
LIN {X 49.4842,Y 134.098,Z 189,A 68.8366,B 1.6928,C -0.0134,E1 1.7556,E2 385.5849} C_DIS
LIN {X 53.0757,Y 132.7162,Z 189,A 67.5469,B 1.6928,C -0.0128,E1 1.7589,E2 386.8433} C_DIS
LIN {X 55.9988,Y 131.5113,Z 189,A 66.2218,B 1.6928,C -0.0109,E1 1.7624,E2 388.1754} C_DIS
LIN {X 58.7181,Y 130.3181,Z 189,A 65.0852,B 1.6928,C -0.0096,E1 1.7653,E2 389.3051} C_DIS
LIN {X 62.0559,Y 128.7624,Z 189,A 63.5984,B 1.6928,C -0.0074,E1 1.769,E2 390.793} C_DIS
LIN {X 65.8162,Y 126.8826,Z 189,A 62.0532,B 1.6928,C -0.0057,E1 1.7728,E2 392.3208} C_DIS
LIN {X 69.5439,Y 124.8792,Z 189,A 60.3969,B 1.6928,C -0.0033,E1 1.7769,E2 393.972} C_DIS
LIN {X 72.7328,Y 123.0493,Z 189,A 58.9283,B 1.6928,C -0.001,E1 1.7804,E2 395.4398} C_DIS
LIN {X 76.4692,Y 120.7624,Z 189,A 57.2174,B 1.6928,C 0.0016,E1 1.7845,E2 397.145} C_DIS
LIN {X 80.2811,Y 118.2625,Z 189,A 55.4812,B 1.6928,C 0.0043,E1 1.7885,E2 398.8699} C_DIS
LIN {X 83.861,Y 115.7513,Z 189,A 53.8583,B 1.6928,C 0.0067,E1 1.7922,E2 400.4766} C_DIS
LIN {X 87.2441,Y 113.224,Z 189,A 52.3323,B 1.6928,C 0.0088,E1 1.7955,E2 401.9818} C_DIS
LIN {X 90.0045,Y 111.0421,Z 189,A 50.974,B 1.6928,C 0.0112,E1 1.7985,E2 403.3336} C_DIS
LIN {X 93.3616,Y 108.2342,Z 189,A 49.2243,B 1.6928,C 0.0146,E1 1.8022,E2 405.0829} C_DIS
LIN {X 96.7579,Y 105.209,Z 189,A 47.5076,B 1.6928,C 0.0176,E1 1.8058,E2 406.7863} C_DIS
LIN {X 100.3156,Y 101.823,Z 189,A 45.7391,B 1.6928,C 0.0205,E1 1.8093,E2 408.5298} C_DIS
LIN {X 103.0331,Y 99.0728,Z 189,A 44.1794,B 1.6928,C 0.0239,E1 1.8123,E2 410.091} C_DIS
LIN {X 106.3852,Y 95.4633,Z 189,A 42.4233,B 1.6927,C 0.0268,E1 1.8156,E2 411.8197} C_DIS
LIN {X 109.2584,Y 92.1617,Z 189,A 40.7749,B 1.6927,C 0.03,E1 1.8186,E2 413.4549} C_DIS
LIN {X 112.029,Y 88.773,Z 189,A 39.1407,B 1.6926,C 0.0333,E1 1.8214,E2 415.0742} C_DIS
LIN {X 114.3807,Y 85.7221,Z 189,A 37.6155,B 1.6926,C 0.0367,E1 1.824,E2 416.5973} C_DIS
LIN {X 116.8663,Y 82.3001,Z 189,A 36.022,B 1.6924,C 0.0401,E1 1.8266,E2 418.1782} C_DIS
LIN {X 119.3281,Y 78.6883,Z 189,A 34.4712,B 1.6924,C 0.043,E1 1.8289,E2 419.7037} C_DIS
LIN {X 121.6902,Y 74.9842,Z 189,A 32.8622,B 1.6923,C 0.0463,E1 1.8313,E2 421.2936} C_DIS
LIN {X 123.8453,Y 71.3684,Z 189,A 31.2833,B 1.6922,C 0.0498,E1 1.8335,E2 422.859} C_DIS
LIN {X 125.7348,Y 67.985,Z 189,A 29.7225,B 1.692,C 0.0537,E1 1.8356,E2 424.4213} C_DIS
LIN {X 127.6002,Y 64.4118,Z 189,A 28.3344,B 1.692,C 0.0563,E1 1.8373,E2 425.7804} C_DIS
LIN {X 129.1367,Y 61.2724,Z 189,A 27.0339,B 1.6919,C 0.0592,E1 1.8389,E2 427.0684} C_DIS
LIN {X 130.5986,Y 58.0908,Z 189,A 25.7127,B 1.6918,C 0.0623,E1 1.8404,E2 428.3794} C_DIS
LIN {X 132.0551,Y 54.7,Z 189,A 24.3591,B 1.6916,C 0.0653,E1 1.8419,E2 429.7172} C_DIS
LIN {X 133.2318,Y 51.7663,Z 189,A 23.1399,B 1.6916,C 0.0683,E1 1.8431,E2 430.9306} C_DIS
LIN {X 134.8006,Y 47.538,Z 189,A 21.3495,B 1.6913,C 0.073,E1 1.8448,E2 432.7196} C_DIS
LIN {X 136.1571,Y 43.4941,Z 189,A 19.9057,B 1.6913,C 0.0758,E1 1.846,E2 434.1292} C_DIS
LIN {X 137.2868,Y 39.787,Z 189,A 18.5281,B 1.6911,C 0.0788,E1 1.8471,E2 435.4844} C_DIS
LIN {X 138.1294,Y 36.7531,Z 189,A 17.322,B 1.6909,C 0.0818,E1 1.848,E2 436.6837} C_DIS
LIN {X 138.9641,Y 33.4589,Z 189,A 16.0485,B 1.6908,C 0.0849,E1 1.8489,E2 437.9461} C_DIS
LIN {X 139.7605,Y 29.9596,Z 189,A 14.733,B 1.6906,C 0.088,E1 1.8496,E2 439.246} C_DIS
LIN {X 140.5217,Y 26.1664,Z 189,A 13.3177,B 1.6904,C 0.0914,E1 1.8504,E2 440.6442} C_DIS
LIN {X 141.0669,Y 23.0416,Z 189,A 12.1295,B 1.6903,C 0.0943,E1 1.8509,E2 441.822} C_DIS
LIN {X 141.5899,Y 19.5775,Z 189,A 10.8359,B 1.6901,C 0.0974,E1 1.8514,E2 443.1016} C_DIS
LIN {X 142.0646,Y 15.7621,Z 189,A 9.3924,B 1.6899,C 0.101,E1 1.8519,E2 444.5329} C_DIS
LIN {X 142.4076,Y 12.2774,Z 189,A 8.1768,B 1.6897,C 0.1036,E1 1.8522,E2 445.7242} C_DIS
LIN {X 142.6458,Y 9.1032,Z 189,A 6.8647,B 1.6895,C 0.1074,E1 1.8525,E2 447.0418} C_DIS
LIN {X 142.8392,Y 5.2611,Z 189,A 5.5479,B 1.6893,C 0.1102,E1 1.8526,E2 448.3293} C_DIS
LIN {X 142.9148,Y 2.4488,Z 189,A 4.4144,B 1.6891,C 0.1134,E1 1.8527,E2 449.4642} C_DIS
LIN {X 142.9313,Y -1.2689,Z 189,A 2.9961,B 1.6889,C 0.117,E1 1.8527,E2 450.8738} C_DIS
LIN {X 142.8389,Y -5.2675,Z 189,A 1.6767,B 1.6887,C 0.1195,E1 1.8526,E2 452.1559} C_DIS
LIN {X 142.6877,Y -8.4241,Z 189,A 0.3683,B 1.6884,C 0.1234,E1 1.8524,E2 453.4706} C_DIS
LIN {X 142.409,Y -12.2608,Z 189,A -0.9422,B 1.6882,C 0.126,E1 1.8521,E2 454.7507} C_DIS
LIN {X 142.1028,Y -15.4073,Z 189,A -2.1587,B 1.688,C 0.1292,E1 1.8518,E2 455.9611} C_DIS
LIN {X 141.6382,Y -19.2257,Z 189,A -3.5754,B 1.6877,C 0.1326,E1 1.8513,E2 457.3619} C_DIS
LIN {X 141.1221,Y -22.7109,Z 189,A -4.901,B 1.6874,C 0.1359,E1 1.8507,E2 458.6767} C_DIS
LIN {X 140.5578,Y -25.9753,Z 189,A -6.108,B 1.6872,C 0.1387,E1 1.8501,E2 459.868} C_DIS
LIN {X 139.8393,Y -29.5946,Z 189,A -7.491,B 1.6869,C 0.1421,E1 1.8494,E2 461.2389} C_DIS
LIN {X 139.0722,Y -33.0105,Z 189,A -8.7826,B 1.6867,C 0.1451,E1 1.8486,E2 462.5162} C_DIS
LIN {X 138.2216,Y -36.4073,Z 189,A -10.158,B 1.6864,C 0.1488,E1 1.8476,E2 463.8886} C_DIS
LIN {X 137.0316,Y -40.6585,Z 189,A -11.7802,B 1.686,C 0.1525,E1 1.8464,E2 465.4918} C_DIS
LIN {X 135.7496,Y -44.7517,Z 189,A -13.3119,B 1.6857,C 0.1558,E1 1.8451,E2 466.9989} C_DIS
LIN {X 134.6959,Y -47.8327,Z 189,A -14.5224,B 1.6855,C 0.1586,E1 1.844,E2 468.1973} C_DIS
LIN {X 133.3584,Y -51.4409,Z 189,A -15.9526,B 1.6851,C 0.1619,E1 1.8426,E2 469.6131} C_DIS
LIN {X 132.1891,Y -54.3792,Z 189,A -17.1285,B 1.6849,C 0.1646,E1 1.8414,E2 470.7772} C_DIS
LIN {X 130.8135,Y -57.6105,Z 189,A -18.4192,B 1.6846,C 0.1675,E1 1.8399,E2 472.0527} C_DIS
LIN {X 129.5872,Y -60.3138,Z 189,A -19.5479,B 1.6843,C 0.1701,E1 1.8386,E2 473.1737} C_DIS
LIN {X 128.0616,Y -63.4883,Z 189,A -20.8745,B 1.684,C 0.1732,E1 1.837,E2 474.4895} C_DIS
LIN {X 126.1472,Y -67.2166,Z 189,A -22.4192,B 1.6837,C 0.1765,E1 1.8351,E2 476.0167} C_DIS
LIN {X 124.2984,Y -70.5764,Z 189,A -23.9375,B 1.6833,C 0.1802,E1 1.833,E2 477.5335} C_DIS
LIN {X 122.0806,Y -74.3476,Z 189,A -25.6143,B 1.6829,C 0.184,E1 1.8306,E2 479.2009} C_DIS
LIN {X 119.4286,Y -78.5356,Z 189,A -27.3899,B 1.6825,C 0.1874,E1 1.8279,E2 480.9484} C_DIS
LIN {X 116.8684,Y -82.2972,Z 189,A -29.0689,B 1.6821,C 0.1908,E1 1.8253,E2 482.6085} C_DIS
LIN {X 114.3945,Y -85.7037,Z 189,A -30.6503,B 1.6818,C 0.194,E1 1.8227,E2 484.1763} C_DIS
LIN {X 112.1423,Y -88.6303,Z 189,A -32.0107,B 1.6815,C 0.1966,E1 1.8204,E2 485.5209} C_DIS
LIN {X 109.8256,Y -91.4852,Z 189,A -33.5111,B 1.681,C 0.2001,E1 1.8177,E2 487.0262} C_DIS
LIN {X 106.6155,Y -95.2061,Z 189,A -35.2887,B 1.6807,C 0.2032,E1 1.8145,E2 488.7781} C_DIS
LIN {X 103.5205,Y -98.5628,Z 189,A -37.0662,B 1.6802,C 0.2068,E1 1.8111,E2 490.5496} C_DIS
LIN {X 100.4508,Y -101.6899,Z 189,A -38.6333,B 1.6799,C 0.2093,E1 1.8081,E2 492.0913} C_DIS
LIN {X 97.2866,Y -104.7204,Z 189,A -40.3785,B 1.6795,C 0.2128,E1 1.8045,E2 493.8362} C_DIS
LIN {X 94.0211,Y -107.6618,Z 189,A -42.0321,B 1.6791,C 0.2156,E1 1.8011,E2 495.4758} C_DIS
LIN {X 90.6777,Y -110.4929,Z 189,A -43.7006,B 1.6787,C 0.2185,E1 1.7975,E2 497.1332} C_DIS
LIN {X 87.249,Y -113.2202,Z 189,A -45.2744,B 1.6785,C 0.2206,E1 1.7941,E2 498.6823} C_DIS
LIN {X 83.8768,Y -115.7398,Z 189,A -46.8795,B 1.6781,C 0.2232,E1 1.7905,E2 500.2768} C_DIS
LIN {X 80.2783,Y -118.2644,Z 189,A -48.5828,B 1.6778,C 0.2259,E1 1.7866,E2 501.9731} C_DIS
LIN {X 76.4723,Y -120.7603,Z 189,A -50.2569,B 1.6775,C 0.2281,E1 1.7827,E2 503.627} C_DIS
LIN {X 73.4895,Y -122.5988,Z 189,A -51.7203,B 1.6771,C 0.2308,E1 1.7792,E2 505.0999} C_DIS
LIN {X 69.8481,Y -124.709,Z 189,A -53.2852,B 1.6768,C 0.2327,E1 1.7754,E2 506.6485} C_DIS
LIN {X 65.9753,Y -126.799,Z 189,A -54.8889,B 1.6766,C 0.2344,E1 1.7715,E2 508.2304} C_DIS
LIN {X 62.8563,Y -128.3734,Z 189,A -56.2444,B 1.6763,C 0.2362,E1 1.7681,E2 509.5805} C_DIS
LIN {X 59.6995,Y -129.8712,Z 189,A -57.588,B 1.6761,C 0.2378,E1 1.7647,E2 510.9168} C_DIS
LIN {X 56.3483,Y -131.3602,Z 189,A -59.0018,B 1.6759,C 0.2395,E1 1.7611,E2 512.3236} C_DIS
LIN {X 53.0832,Y -132.7132,Z 189,A -60.2945,B 1.6757,C 0.2406,E1 1.7578,E2 513.5993} C_DIS
LIN {X 50.1245,Y -133.8582,Z 189,A -61.6401,B 1.6754,C 0.2426,E1 1.7542,E2 514.9564} C_DIS
LIN {X 46.5042,Y -135.159,Z 189,A -63.0378,B 1.6753,C 0.2436,E1 1.7506,E2 516.3343} C_DIS
LIN {X 43.1397,Y -136.2703,Z 189,A -64.4834,B 1.675,C 0.2453,E1 1.7467,E2 517.7845} C_DIS
LIN {X 38.7797,Y -137.5745,Z 189,A -66.336,B 1.6747,C 0.2473,E1 1.7417,E2 519.6424} C_DIS
LIN {X 35.0816,Y -138.5634,Z 189,A -67.7178,B 1.6747,C 0.2479,E1 1.738,E2 521.0031} C_DIS
LIN {X 31.6853,Y -139.3793,Z 189,A -69.0813,B 1.6745,C 0.249,E1 1.7343,E2 522.3622} C_DIS
LIN {X 28.2652,Y -140.1131,Z 189,A -70.4812,B 1.6743,C 0.2502,E1 1.7305,E2 523.7626} C_DIS
LIN {X 24.7745,Y -140.7727,Z 189,A -71.8381,B 1.6743,C 0.2509,E1 1.7268,E2 525.1106} C_DIS
LIN {X 21.3169,Y -141.3381,Z 189,A -73.2101,B 1.6741,C 0.2517,E1 1.723,E2 526.4788} C_DIS
LIN {X 17.8454,Y -141.8191,Z 189,A -74.6822,B 1.6739,C 0.2529,E1 1.7189,E2 527.9615} C_DIS
LIN {X 14.0273,Y -142.2461,Z 189,A -76.1205,B 1.6739,C 0.2533,E1 1.7149,E2 529.3858} C_DIS
LIN {X 10.8564,Y -142.5235,Z 189,A -77.3806,B 1.6738,C 0.2539,E1 1.7114,E2 530.6443} C_DIS
LIN {X 7.0168,Y -142.7634,Z 189,A -78.8867,B 1.6737,C 0.2544,E1 1.7072,E2 532.146} C_DIS
LIN {X 3.8569,Y -142.8837,Z 189,A -80.1411,B 1.6737,C 0.2548,E1 1.7036,E2 533.3992} C_DIS
LIN {X 1.0097,Y -142.9296,Z 189,A -80.9142,B 1.6738,C 0.2534,E1 1.7016,E2 534.1192} C_DIS
Enddeposition()
LIN {X 0.9699,Y -133.9666,Z 190,A -77.995,B 1.0116,C 0.2061,E1 1.046,E2 530.7026} C_DIS
Startdeposition()
$VEL.CP = VEL_PRINT
LIN {X 3.2812,Y -133.9326,Z 190,A -76.7854,B 1.0119,C 0.2049,E1 1.0495,E2 529.4615} C_DIS
LIN {X 6.556,Y -133.8116,Z 190,A -75.3807,B 1.012,C 0.2041,E1 1.0534,E2 528.0555} C_DIS
LIN {X 10.1305,Y -133.5889,Z 190,A -73.9566,B 1.0122,C 0.2035,E1 1.0574,E2 526.6458} C_DIS
LIN {X 13.1178,Y -133.3285,Z 190,A -72.6917,B 1.0123,C 0.2027,E1 1.061,E2 525.3825} C_DIS
LIN {X 16.6351,Y -132.9373,Z 190,A -71.2609,B 1.0125,C 0.2018,E1 1.0649,E2 523.9626} C_DIS
LIN {X 19.878,Y -132.4904,Z 190,A -69.8709,B 1.0127,C 0.2007,E1 1.0688,E2 522.5731} C_DIS
LIN {X 22.9045,Y -132.0012,Z 190,A -68.6324,B 1.0129,C 0.1998,E1 1.0722,E2 521.344} C_DIS
LIN {X 26.1312,Y -131.3999,Z 190,A -67.2927,B 1.0131,C 0.1988,E1 1.0759,E2 520.0124} C_DIS
LIN {X 29.3427,Y -130.7199,Z 190,A -65.9561,B 1.0133,C 0.1976,E1 1.0796,E2 518.6843} C_DIS
LIN {X 32.5383,Y -129.961,Z 190,A -64.6169,B 1.0136,C 0.1964,E1 1.0832,E2 517.3533} C_DIS
LIN {X 35.7324,Y -129.1191,Z 190,A -63.2828,B 1.0138,C 0.1951,E1 1.0869,E2 516.0294} C_DIS
LIN {X 39.1553,Y -128.1221,Z 190,A -61.8429,B 1.0141,C 0.1937,E1 1.0907,E2 514.6003} C_DIS
LIN {X 42.0215,Y -127.2112,Z 190,A -60.6242,B 1.0143,C 0.1923,E1 1.094,E2 513.3901} C_DIS
LIN {X 45.1444,Y -126.1367,Z 190,A -59.3034,B 1.0146,C 0.1909,E1 1.0974,E2 512.0812} C_DIS
LIN {X 48.2129,Y -124.996,Z 190,A -57.9904,B 1.0149,C 0.1894,E1 1.1009,E2 510.7794} C_DIS
LIN {X 51.5062,Y -123.6749,Z 190,A -56.5699,B 1.0152,C 0.1876,E1 1.1045,E2 509.3713} C_DIS
LIN {X 54.2546,Y -122.495,Z 190,A -55.381,B 1.0155,C 0.1861,E1 1.1076,E2 508.1942} C_DIS
LIN {X 57.5279,Y -120.9915,Z 190,A -53.9384,B 1.0158,C 0.1842,E1 1.1112,E2 506.7641} C_DIS
LIN {X 60.4859,Y -119.5404,Z 190,A -52.7191,B 1.0161,C 0.1828,E1 1.1142,E2 505.5701} C_DIS
LIN {X 63.1521,Y -118.1558,Z 190,A -51.4422,B 1.0165,C 0.1808,E1 1.1174,E2 504.2935} C_DIS
LIN {X 66.0292,Y -116.5727,Z 190,A -50.1352,B 1.0168,C 0.1789,E1 1.1206,E2 502.999} C_DIS
LIN {X 68.8858,Y -114.9076,Z 190,A -48.8303,B 1.0171,C 0.177,E1 1.1237,E2 501.7081} C_DIS
LIN {X 71.9144,Y -113.0369,Z 190,A -47.465,B 1.0175,C 0.175,E1 1.1269,E2 500.3634} C_DIS
LIN {X 74.4273,Y -111.3978,Z 190,A -46.2537,B 1.0178,C 0.173,E1 1.1298,E2 499.1611} C_DIS
LIN {X 77.3581,Y -109.383,Z 190,A -44.8574,B 1.0182,C 0.1708,E1 1.1329,E2 497.7807} C_DIS
LIN {X 80.0135,Y -107.4557,Z 190,A -43.497,B 1.0186,C 0.1683,E1 1.136,E2 496.4252} C_DIS
LIN {X 83.6094,Y -104.6824,Z 190,A -41.767,B 1.0191,C 0.1655,E1 1.1398,E2 494.723} C_DIS
LIN {X 86.8598,Y -102.0013,Z 190,A -40.0525,B 1.0196,C 0.1623,E1 1.1434,E2 493.0191} C_DIS
LIN {X 89.9078,Y -99.3252,Z 190,A -38.4656,B 1.02,C 0.1594,E1 1.1467,E2 491.4511} C_DIS
LIN {X 93.4068,Y -96.0424,Z 190,A -36.6489,B 1.0205,C 0.1562,E1 1.1503,E2 489.665} C_DIS
LIN {X 96.4891,Y -92.9454,Z 190,A -34.9125,B 1.0211,C 0.1527,E1 1.1537,E2 487.9452} C_DIS
LIN {X 99.0396,Y -90.2226,Z 190,A -33.5034,B 1.0214,C 0.1501,E1 1.1564,E2 486.5603} C_DIS
LIN {X 101.9987,Y -86.8629,Z 190,A -31.7699,B 1.0219,C 0.1467,E1 1.1595,E2 484.8499} C_DIS
LIN {X 104.6848,Y -83.6063,Z 190,A -30.1429,B 1.0224,C 0.1434,E1 1.1623,E2 483.2457} C_DIS
LIN {X 107.5874,Y -79.8366,Z 190,A -28.4219,B 1.0229,C 0.1402,E1 1.1652,E2 481.5656} C_DIS
LIN {X 109.6445,Y -76.9874,Z 190,A -26.994,B 1.0233,C 0.137,E1 1.1675,E2 480.1466} C_DIS
LIN {X 111.5538,Y -74.1937,Z 190,A -25.8243,B 1.0236,C 0.1349,E1 1.1692,E2 479.013} C_DIS
LIN {X 113.3364,Y -71.4405,Z 190,A -24.5287,B 1.0239,C 0.132,E1 1.1712,E2 477.7308} C_DIS
LIN {X 115.0513,Y -68.6447,Z 190,A -23.2431,B 1.0243,C 0.1291,E1 1.173,E2 476.4597} C_DIS
LIN {X 116.678,Y -65.8421,Z 190,A -21.9601,B 1.0247,C 0.1261,E1 1.1748,E2 475.1894} C_DIS
LIN {X 118.2872,Y -62.9044,Z 190,A -20.807,B 1.0249,C 0.124,E1 1.1763,E2 474.0725} C_DIS
LIN {X 119.9299,Y -59.7111,Z 190,A -19.5101,B 1.0253,C 0.1213,E1 1.1779,E2 472.8061} C_DIS
LIN {X 121.1116,Y -57.2765,Z 190,A -18.3539,B 1.0256,C 0.1183,E1 1.1793,E2 471.6492} C_DIS
LIN {X 122.4787,Y -54.2911,Z 190,A -17.123,B 1.0259,C 0.1156,E1 1.1806,E2 470.4402} C_DIS
LIN {X 123.8879,Y -50.9962,Z 190,A -15.7647,B 1.0263,C 0.1125,E1 1.1821,E2 469.1038} C_DIS
LIN {X 125.2107,Y -47.6566,Z 190,A -14.4431,B 1.0266,C 0.1095,E1 1.1834,E2 467.8094} C_DIS
LIN {X 126.2318,Y -44.8806,Z 190,A -13.2254,B 1.0269,C 0.1064,E1 1.1846,E2 466.597} C_DIS
LIN {X 127.6232,Y -40.7519,Z 190,A -11.5728,B 1.0273,C 0.1025,E1 1.186,E2 464.9706} C_DIS
LIN {X 128.7362,Y -37.0908,Z 190,A -10.192,B 1.0276,C 0.0995,E1 1.187,E2 463.622} C_DIS
LIN {X 129.6196,Y -33.8765,Z 190,A -8.9374,B 1.0279,C 0.0965,E1 1.1879,E2 462.3888} C_DIS
LIN {X 130.4638,Y -30.4634,Z 190,A -7.6631,B 1.0282,C 0.0936,E1 1.1888,E2 461.1431} C_DIS
LIN {X 131.1284,Y -27.4654,Z 190,A -6.4397,B 1.0284,C 0.0905,E1 1.1895,E2 459.9305} C_DIS
LIN {X 131.7613,Y -24.2453,Z 190,A -5.2047,B 1.0287,C 0.0876,E1 1.1901,E2 458.7164} C_DIS
LIN {X 132.2722,Y -21.2864,Z 190,A -3.9972,B 1.029,C 0.0844,E1 1.1906,E2 457.518} C_DIS
LIN {X 132.7534,Y -18.0384,Z 190,A -2.8287,B 1.0292,C 0.0818,E1 1.1911,E2 456.3787} C_DIS
LIN {X 133.1848,Y -14.5023,Z 190,A -1.5151,B 1.0294,C 0.0787,E1 1.1915,E2 455.091} C_DIS
LIN {X 133.5426,Y -10.7312,Z 190,A 0.0926,B 1.0297,C 0.0742,E1 1.1919,E2 453.484} C_DIS
LIN {X 133.8243,Y -6.3036,Z 190,A 1.5867,B 1.03,C 0.0711,E1 1.1921,E2 452.04} C_DIS
LIN {X 133.9402,Y -3.0054,Z 190,A 2.9196,B 1.0302,C 0.0676,E1 1.1922,E2 450.7163} C_DIS
LIN {X 133.974,Y -0.0071,Z 190,A 4.1166,B 1.0304,C 0.0645,E1 1.1922,E2 449.5293} C_DIS
LIN {X 133.9323,Y 3.2916,Z 190,A 5.2247,B 1.0305,C 0.0622,E1 1.1922,E2 448.4586} C_DIS
LIN {X 133.8109,Y 6.5705,Z 190,A 6.4923,B 1.0307,C 0.059,E1 1.192,E2 447.2072} C_DIS
LIN {X 133.5896,Y 10.1212,Z 190,A 7.7798,B 1.0309,C 0.056,E1 1.1918,E2 445.9482} C_DIS
LIN {X 133.329,Y 13.1131,Z 190,A 8.9357,B 1.031,C 0.0531,E1 1.1915,E2 444.8077} C_DIS
LIN {X 132.931,Y 16.6833,Z 190,A 10.3214,B 1.0312,C 0.0496,E1 1.191,E2 443.4401} C_DIS
LIN {X 132.4819,Y 19.9331,Z 190,A 11.5345,B 1.0314,C 0.0467,E1 1.1905,E2 442.2498} C_DIS
LIN {X 132.0026,Y 22.8966,Z 190,A 12.6532,B 1.0314,C 0.0441,E1 1.19,E2 441.1509} C_DIS
LIN {X 131.3984,Y 26.1386,Z 190,A 13.8917,B 1.0316,C 0.0411,E1 1.1894,E2 439.933} C_DIS
LIN {X 130.7167,Y 29.3567,Z 190,A 15.1296,B 1.0317,C 0.0381,E1 1.1887,E2 438.7151} C_DIS
LIN {X 129.9573,Y 32.5527,Z 190,A 16.3673,B 1.0318,C 0.0351,E1 1.1878,E2 437.4973} C_DIS
LIN {X 129.1199,Y 35.7295,Z 190,A 17.6775,B 1.0319,C 0.0318,E1 1.1869,E2 436.198} C_DIS
LIN {X 128.12,Y 39.1621,Z 190,A 18.956,B 1.032,C 0.029,E1 1.1859,E2 434.9494} C_DIS
LIN {X 127.2096,Y 42.0262,Z 190,A 20.0921,B 1.032,C 0.0263,E1 1.1849,E2 433.831} C_DIS
LIN {X 126.0036,Y 45.5135,Z 190,A 21.4097,B 1.0321,C 0.0234,E1 1.1837,E2 432.5442} C_DIS
LIN {X 124.9915,Y 48.2245,Z 190,A 22.5803,B 1.0322,C 0.0204,E1 1.1826,E2 431.3812} C_DIS
LIN {X 123.6656,Y 51.5286,Z 190,A 23.9295,B 1.0322,C 0.0173,E1 1.1812,E2 430.0523} C_DIS
LIN {X 122.3493,Y 54.5805,Z 190,A 25.1795,B 1.0323,C 0.0144,E1 1.1798,E2 428.8223} C_DIS
LIN {X 120.9967,Y 57.517,Z 190,A 26.4191,B 1.0323,C 0.0115,E1 1.1783,E2 427.5994} C_DIS
LIN {X 119.5394,Y 60.4879,Z 190,A 27.5882,B 1.0323,C 0.0091,E1 1.1769,E2 426.4591} C_DIS
LIN {X 118.1527,Y 63.1578,Z 190,A 28.8142,B 1.0323,C 0.0061,E1 1.1753,E2 425.2401} C_DIS
LIN {X 116.5687,Y 66.0362,Z 190,A 30.1241,B 1.0324,C 0.0031,E1 1.1736,E2 423.9411} C_DIS
LIN {X 114.9088,Y 68.8838,Z 190,A 31.352,B 1.0324,C 0.0004,E1 1.1718,E2 422.7342} C_DIS
LIN {X 113.0412,Y 71.9077,Z 190,A 32.6477,B 1.0324,C -0.0023,E1 1.1699,E2 421.4645} C_DIS
LIN {X 111.4035,Y 74.4187,Z 190,A 33.823,B 1.0324,C -0.0049,E1 1.1681,E2 420.3014} C_DIS
LIN {X 109.3745,Y 77.3701,Z 190,A 35.3079,B 1.0324,C -0.0084,E1 1.1658,E2 418.8217} C_DIS
LIN {X 106.6208,Y 81.1234,Z 190,A 37.006,B 1.0324,C -0.0117,E1 1.163,E2 417.1574} C_DIS
LIN {X 104.0786,Y 84.3602,Z 190,A 38.5747,B 1.0324,C -0.0149,E1 1.1603,E2 415.6106} C_DIS
LIN {X 101.4457,Y 87.5081,Z 190,A 40.2461,B 1.0322,C -0.0186,E1 1.1573,E2 413.9486} C_DIS
LIN {X 98.6231,Y 90.6773,Z 190,A 41.8771,B 1.0322,C -0.0218,E1 1.1542,E2 412.3386} C_DIS
LIN {X 95.8001,Y 93.6551,Z 190,A 43.461,B 1.0322,C -0.0249,E1 1.1512,E2 410.7741} C_DIS
LIN {X 92.3722,Y 97.0378,Z 190,A 45.334,B 1.032,C -0.0285,E1 1.1475,E2 408.9223} C_DIS
LIN {X 89.2525,Y 99.9146,Z 190,A 46.9757,B 1.032,C -0.0315,E1 1.1441,E2 407.3001} C_DIS
LIN {X 85.7359,Y 102.9484,Z 190,A 48.7199,B 1.0318,C -0.0345,E1 1.1404,E2 405.5833} C_DIS
LIN {X 82.4326,Y 105.6121,Z 190,A 50.3217,B 1.0318,C -0.0372,E1 1.1369,E2 404.0055} C_DIS
LIN {X 79.8197,Y 107.6,Z 190,A 51.6166,B 1.0317,C -0.0394,E1 1.134,E2 402.723} C_DIS
LIN {X 76.9087,Y 109.7,Z 190,A 53.0071,B 1.0316,C -0.0417,E1 1.1309,E2 401.3487} C_DIS
LIN {X 74.1974,Y 111.5513,Z 190,A 54.297,B 1.0315,C -0.0438,E1 1.1279,E2 400.0716} C_DIS
LIN {X 71.4314,Y 113.3422,Z 190,A 55.584,B 1.0314,C -0.0459,E1 1.1249,E2 398.7982} C_DIS
LIN {X 68.6415,Y 115.0532,Z 190,A 56.9187,B 1.0313,C -0.048,E1 1.1217,E2 397.4709} C_DIS
LIN {X 65.8118,Y 116.6951,Z 190,A 58.1597,B 1.0313,C -0.0498,E1 1.1187,E2 396.2475} C_DIS
LIN {X 62.9452,Y 118.2658,Z 190,A 59.4313,B 1.0311,C -0.0516,E1 1.1156,E2 394.99} C_DIS
LIN {X 60.0106,Y 119.7821,Z 190,A 60.7693,B 1.0311,C -0.0536,E1 1.1123,E2 393.6604} C_DIS
LIN {X 57.2801,Y 121.1099,Z 190,A 61.995,B 1.0309,C -0.0553,E1 1.1092,E2 392.4428} C_DIS
LIN {X 54.2813,Y 122.4831,Z 190,A 63.2906,B 1.0309,C -0.0569,E1 1.1059,E2 391.16} C_DIS
LIN {X 50.9411,Y 123.9109,Z 190,A 64.7414,B 1.0307,C -0.0588,E1 1.1021,E2 389.7208} C_DIS
LIN {X 47.9647,Y 125.0925,Z 190,A 66.0233,B 1.0307,C -0.0604,E1 1.0988,E2 388.4487} C_DIS
LIN {X 44.7818,Y 126.2674,Z 190,A 67.381,B 1.0306,C -0.0619,E1 1.0952,E2 387.1014} C_DIS
LIN {X 42.0467,Y 127.2028,Z 190,A 68.5465,B 1.0305,C -0.0632,E1 1.0921,E2 385.9438} C_DIS
LIN {X 38.6263,Y 128.2839,Z 190,A 69.994,B 1.0304,C -0.0648,E1 1.0882,E2 384.5061} C_DIS
LIN {X 35.4567,Y 129.1961,Z 190,A 71.327,B 1.0303,C -0.0661,E1 1.0847,E2 383.1819} C_DIS
LIN {X 32.2795,Y 130.0267,Z 190,A 72.6583,B 1.0303,C -0.0674,E1 1.081,E2 381.8588} C_DIS
LIN {X 29.0832,Y 130.7791,Z 190,A 74.1221,B 1.0301,C -0.069,E1 1.077,E2 380.3889} C_DIS
LIN {X 25.8658,Y 131.4531,Z 190,A 75.4251,B 1.0301,C -0.07,E1 1.0734,E2 379.0974} C_DIS
LIN {X 22.9065,Y 132.0009,Z 190,A 76.5635,B 1.03,C -0.0707,E1 1.0703,E2 377.9754} C_DIS
LIN {X 19.3761,Y 132.564,Z 190,A 77.9623,B 1.03,C -0.0716,E1 1.0664,E2 376.591} C_DIS
LIN {X 16.4012,Y 132.9652,Z 190,A 79.356,B 1.0298,C -0.0729,E1 1.0625,E2 375.186} C_DIS
LIN {X 13.1383,Y 133.3266,Z 190,A 80.6421,B 1.0298,C -0.0736,E1 1.0589,E2 373.913} C_DIS
LIN {X 9.8674,Y 133.6081,Z 190,A 82.0408,B 1.0298,C -0.0745,E1 1.055,E2 372.5153} C_DIS
LIN {X 6.3162,Y 133.8236,Z 190,A 83.5275,B 1.0297,C -0.0753,E1 1.0508,E2 371.0329} C_DIS
LIN {X 3.0078,Y 133.9402,Z 190,A 84.8269,B 1.0297,C -0.0757,E1 1.0472,E2 369.7465} C_DIS
LIN {X -0.2712,Y 133.9726,Z 190,A 86.1584,B 1.0297,C -0.0761,E1 1.0434,E2 368.423} C_DIS
LIN {X -3.2732,Y 133.9328,Z 190,A 87.5698,B 1.0295,C -0.0769,E1 1.0394,E2 366.9985} C_DIS
LIN {X -6.5692,Y 133.8109,Z 190,A 88.9281,B 1.0295,C -0.0772,E1 1.0356,E2 365.6463} C_DIS
LIN {X -10.5568,Y 133.5573,Z 190,A 90.5304,B 1.0295,C -0.0774,E1 1.0311,E2 364.0562} C_DIS
LIN {X -13.129,Y 133.3274,Z 190,A 91.6776,B 1.0295,C -0.0776,E1 1.0279,E2 362.9048} C_DIS
LIN {X -16.6633,Y 132.9337,Z 190,A 93.1504,B 1.0295,C -0.0776,E1 1.0237,E2 361.4379} C_DIS
LIN {X -19.9154,Y 132.4846,Z 190,A 94.5884,B 1.0295,C -0.0778,E1 1.0197,E2 359.9968} C_DIS
LIN {X -22.8763,Y 132.0063,Z 190,A 95.9525,B 1.0295,C -0.0778,E1 1.0159,E2 358.6247} C_DIS
LIN {X -26.1361,Y 131.3989,Z 190,A 97.2979,B 1.0295,C -0.0776,E1 1.0122,E2 357.2877} C_DIS
LIN {X -29.349,Y 130.7184,Z 190,A 98.7122,B 1.0295,C -0.0774,E1 1.0083,E2 355.873} C_DIS
LIN {X -32.5444,Y 129.9594,Z 190,A 100.1328,B 1.0295,C -0.0771,E1 1.0044,E2 354.4513} C_DIS
LIN {X -35.7201,Y 129.1225,Z 190,A 101.6429,B 1.0295,C -0.0768,E1 1.0002,E2 352.9306} C_DIS
LIN {X -39.1576,Y 128.1213,Z 190,A 103.1195,B 1.0296,C -0.0761,E1 0.9962,E2 351.4606} C_DIS
LIN {X -42.5995,Y 127.0187,Z 190,A 104.5822,B 1.0296,C -0.0753,E1 0.9923,E2 350.0075} C_DIS
LIN {X -45.142,Y 126.1375,Z 190,A 105.8831,B 1.0296,C -0.0749,E1 0.9888,E2 348.6912} C_DIS
LIN {X -48.2185,Y 124.9938,Z 190,A 107.3744,B 1.0297,C -0.0741,E1 0.9849,E2 347.1914} C_DIS
LIN {X -51.524,Y 123.6675,Z 190,A 108.9069,B 1.0298,C -0.0731,E1 0.9809,E2 345.6586} C_DIS
LIN {X -54.2827,Y 122.4824,Z 190,A 110.3146,B 1.0298,C -0.0723,E1 0.9772,E2 344.2384} C_DIS
LIN {X -57.597,Y 120.9585,Z 190,A 111.842,B 1.03,C -0.071,E1 0.9733,E2 342.7154} C_DIS
LIN {X -60.5099,Y 119.5282,Z 190,A 113.2152,B 1.03,C -0.0698,E1 0.9698,E2 341.3444} C_DIS
LIN {X -63.1565,Y 118.1534,Z 190,A 114.6607,B 1.0301,C -0.0687,E1 0.9662,E2 339.8816} C_DIS
LIN {X -66.0444,Y 116.5641,Z 190,A 116.1442,B 1.0302,C -0.0674,E1 0.9625,E2 338.391} C_DIS
LIN {X -69.538,Y 114.5138,Z 190,A 118.1018,B 1.0303,C -0.0656,E1 0.9577,E2 336.41} C_DIS
LIN {X -73.0619,Y 112.2981,Z 190,A 119.8725,B 1.0305,C -0.0635,E1 0.9535,E2 334.6414} C_DIS
LIN {X -75.7909,Y 110.4746,Z 190,A 121.4238,B 1.0305,C -0.0619,E1 0.9498,E2 333.0749} C_DIS
LIN {X -78.9395,Y 108.2479,Z 190,A 123.1041,B 1.0307,C -0.0597,E1 0.946,E2 331.3923} C_DIS
LIN {X -81.7835,Y 106.1153,Z 190,A 124.9207,B 1.0307,C -0.0577,E1 0.9418,E2 329.5443} C_DIS
LIN {X -85.2777,Y 103.3279,Z 190,A 126.9345,B 1.031,C -0.0549,E1 0.9374,E2 327.5205} C_DIS
LIN {X -88.123,Y 100.912,Z 190,A 128.5972,B 1.031,C -0.0524,E1 0.9339,E2 325.8515} C_DIS
LIN {X -90.6699,Y 98.6299,Z 190,A 130.2986,B 1.0312,C -0.0501,E1 0.9303,E2 324.1247} C_DIS
LIN {X -93.67,Y 95.7855,Z 190,A 132.2286,B 1.0313,C -0.0471,E1 0.9263,E2 322.1779} C_DIS
LIN {X -96.557,Y 92.8752,Z 190,A 134.1791,B 1.0315,C -0.044,E1 0.9225,E2 320.2067} C_DIS
LIN {X -99.2596,Y 89.9802,Z 190,A 135.9147,B 1.0316,C -0.0409,E1 0.9191,E2 318.4675} C_DIS
LIN {X -101.5224,Y 87.4191,Z 190,A 137.6137,B 1.0317,C -0.0381,E1 0.916,E2 316.7429} C_DIS
LIN {X -104.1728,Y 84.2434,Z 190,A 139.6005,B 1.0318,C -0.0346,E1 0.9124,E2 314.7328} C_DIS
LIN {X -106.6187,Y 81.1261,Z 190,A 141.3616,B 1.0319,C -0.0311,E1 0.9093,E2 312.9653} C_DIS
LIN {X -108.5737,Y 78.4899,Z 190,A 142.9765,B 1.032,C -0.0281,E1 0.9066,E2 311.3275} C_DIS
LIN {X -110.6374,Y 75.5536,Z 190,A 144.6502,B 1.0321,C -0.0248,E1 0.9039,E2 309.6391} C_DIS
LIN {X -112.3023,Y 73.0554,Z 190,A 146.1999,B 1.0321,C -0.0219,E1 0.9015,E2 308.06} C_DIS
LIN {X -114.2059,Y 70.0422,Z 190,A 147.8097,B 1.0322,C -0.0184,E1 0.8991,E2 306.4414} C_DIS
LIN {X -115.893,Y 67.2139,Z 190,A 149.3968,B 1.0323,C -0.0151,E1 0.8968,E2 304.8348} C_DIS
LIN {X -117.5033,Y 64.3577,Z 190,A 151.0021,B 1.0323,C -0.0117,E1 0.8946,E2 303.2071} C_DIS
LIN {X -118.9152,Y 61.7084,Z 190,A 152.464,B 1.0323,C -0.0086,E1 0.8927,E2 301.7255} C_DIS
LIN {X -120.3837,Y 58.7912,Z 190,A 154.1909,B 1.0324,C -0.005,E1 0.8905,E2 299.9612} C_DIS
LIN {X -121.9278,Y 55.521,Z 190,A 155.8043,B 1.0324,C -0.0012,E1 0.8886,E2 298.3411} C_DIS
LIN {X -123.1383,Y 52.7778,Z 190,A 157.2992,B 1.0324,C 0.0022,E1 0.8869,E2 296.8222} C_DIS
LIN {X -124.5009,Y 49.4805,Z 190,A 159.0856,B 1.0324,C 0.0062,E1 0.885,E2 295.0063} C_DIS
LIN {X -125.6749,Y 46.4174,Z 190,A 160.6297,B 1.0324,C 0.0099,E1 0.8835,E2 293.4464} C_DIS
LIN {X -126.7744,Y 43.3241,Z 190,A 162.2218,B 1.0324,C 0.0137,E1 0.882,E2 291.8331} C_DIS
LIN {X -127.7137,Y 40.4685,Z 190,A 163.7557,B 1.0323,C 0.0172,E1 0.8806,E2 290.2705} C_DIS
LIN {X -128.768,Y 36.9821,Z 190,A 165.5191,B 1.0322,C 0.0215,E1 0.8792,E2 288.4836} C_DIS
LIN {X -129.6059,Y 33.9276,Z 190,A 167.0773,B 1.0322,C 0.0253,E1 0.8781,E2 286.9019} C_DIS
LIN {X -130.5312,Y 30.1686,Z 190,A 168.788,B 1.032,C 0.0298,E1 0.877,E2 285.1857} C_DIS
LIN {X -131.1277,Y 27.4688,Z 190,A 170.384,B 1.0319,C 0.0334,E1 0.876,E2 283.5408} C_DIS
LIN {X -131.7611,Y 24.2463,Z 190,A 172.0285,B 1.0317,C 0.0374,E1 0.8751,E2 281.868} C_DIS
LIN {X -132.2723,Y 21.2855,Z 190,A 173.6015,B 1.0316,C 0.0412,E1 0.8744,E2 280.2607} C_DIS
LIN {X -132.8336,Y 17.4269,Z 190,A 175.233,B 1.0314,C 0.0458,E1 0.8738,E2 278.6346} C_DIS
LIN {X -133.1868,Y 14.4829,Z 190,A 176.9595,B 1.0312,C 0.0497,E1 0.8732,E2 276.8527} C_DIS
LIN {X -133.4784,Y 11.4914,Z 190,A 178.401,B 1.031,C 0.0534,E1 0.8728,E2 275.3927} C_DIS
LIN {X -133.7369,Y 7.9388,Z 190,A -179.8442,B 1.0308,C 0.0579,E1 0.8725,E2 273.6103} C_DIS
LIN {X -133.8925,Y 4.6489,Z 190,A -178.2172,B 1.0305,C 0.062,E1 0.8723,E2 271.957} C_DIS
LIN {X -133.9682,Y 1.0775,Z 190,A -176.6248,B 1.0303,C 0.0663,E1 0.8723,E2 270.3574} C_DIS
LIN {X -133.9632,Y -1.6468,Z 190,A -175.0375,B 1.03,C 0.07,E1 0.8723,E2 268.718} C_DIS
LIN {X -133.8816,Y -4.9301,Z 190,A -173.4159,B 1.0298,C 0.0741,E1 0.8724,E2 267.07} C_DIS
LIN {X -133.703,Y -8.4891,Z 190,A -171.6623,B 1.0294,C 0.0785,E1 0.8727,E2 265.2883} C_DIS
LIN {X -133.3956,Y -12.4192,Z 190,A -169.4991,B 1.029,C 0.0836,E1 0.8732,E2 263.0654} C_DIS
LIN {X -132.9277,Y -16.7085,Z 190,A -167.601,B 1.0286,C 0.0888,E1 0.8738,E2 261.1615} C_DIS
LIN {X -132.482,Y -19.9323,Z 190,A -165.9231,B 1.0282,C 0.0928,E1 0.8745,E2 259.4478} C_DIS
LIN {X -132.001,Y -22.9059,Z 190,A -164.4271,B 1.0279,C 0.0965,E1 0.8752,E2 257.9258} C_DIS
LIN {X -131.3975,Y -26.1433,Z 190,A -162.8025,B 1.0275,C 0.1005,E1 0.8761,E2 256.2741} C_DIS
LIN {X -130.7165,Y -29.3572,Z 190,A -161.1795,B 1.0271,C 0.1044,E1 0.8771,E2 254.6235} C_DIS
LIN {X -129.957,Y -32.5538,Z 190,A -159.5459,B 1.0267,C 0.1084,E1 0.8782,E2 252.9609} C_DIS
LIN {X -129.1145,Y -35.7486,Z 190,A -157.9333,B 1.0263,C 0.1122,E1 0.8794,E2 251.323} C_DIS
LIN {X -128.1272,Y -39.1385,Z 190,A -156.1951,B 1.0258,C 0.1163,E1 0.8808,E2 249.5556} C_DIS
LIN {X -127.2271,Y -41.9737,Z 190,A -154.7385,B 1.0254,C 0.1198,E1 0.8821,E2 248.0754} C_DIS
LIN {X -126.1865,Y -45.0063,Z 190,A -153.1852,B 1.025,C 0.1234,E1 0.8835,E2 246.4987} C_DIS
LIN {X -124.9941,Y -48.218,Z 190,A -151.4769,B 1.0245,C 0.1272,E1 0.8853,E2 244.7589} C_DIS
LIN {X -123.6669,Y -51.5255,Z 190,A -149.7332,B 1.0241,C 0.1311,E1 0.8871,E2 242.9867} C_DIS
LIN {X -122.4811,Y -54.2857,Z 190,A -148.1871,B 1.0236,C 0.1344,E1 0.8889,E2 241.4063} C_DIS
LIN {X -120.9875,Y -57.5363,Z 190,A -146.5272,B 1.0231,C 0.1381,E1 0.8909,E2 239.7297} C_DIS
LIN {X -119.5397,Y -60.4872,Z 190,A -144.9433,B 1.0227,C 0.1416,E1 0.8929,E2 238.1224} C_DIS
LIN {X -118.1484,Y -63.166,Z 190,A -143.47,B 1.0222,C 0.1446,E1 0.8949,E2 236.6252} C_DIS
LIN {X -116.566,Y -66.0411,Z 190,A -141.7392,B 1.0218,C 0.1479,E1 0.8973,E2 234.8508} C_DIS
LIN {X -114.3189,Y -69.858,Z 190,A -139.5866,B 1.0211,C 0.1522,E1 0.9005,E2 232.6638} C_DIS
LIN {X -112.305,Y -73.0514,Z 190,A -137.7962,B 1.0206,C 0.1557,E1 0.9032,E2 230.85} C_DIS
LIN {X -109.6858,Y -76.9288,Z 190,A -135.56,B 1.0199,C 0.16,E1 0.9068,E2 228.5823} C_DIS
LIN {X -107.4354,Y -80.0408,Z 190,A -133.7572,B 1.0194,C 0.1633,E1 0.9099,E2 226.758} C_DIS
LIN {X -104.6837,Y -83.6077,Z 190,A -131.6059,B 1.0188,C 0.1671,E1 0.9136,E2 224.5763} C_DIS
LIN {X -101.982,Y -86.8825,Z 190,A -129.7077,B 1.0182,C 0.1706,E1 0.9171,E2 222.6671} C_DIS
LIN {X -99.7273,Y -89.4615,Z 190,A -128.0938,B 1.0178,C 0.1732,E1 0.9201,E2 221.033} C_DIS
LIN {X -97.0242,Y -92.3864,Z 190,A -126.1664,B 1.0173,C 0.1762,E1 0.9239,E2 219.0749} C_DIS
LIN {X -94.1715,Y -95.293,Z 190,A -124.2954,B 1.0168,C 0.1791,E1 0.9276,E2 217.1862} C_DIS
LIN {X -91.2396,Y -98.1031,Z 190,A -122.304,B 1.0163,C 0.1818,E1 0.9318,E2 215.1597} C_DIS
LIN {X -88.1298,Y -100.906,Z 190,A -120.354,B 1.0158,C 0.1845,E1 0.936,E2 213.1877} C_DIS
LIN {X -84.889,Y -103.6474,Z 190,A -118.3976,B 1.0153,C 0.187,E1 0.9402,E2 211.2116} C_DIS
LIN {X -81.6739,Y -106.1998,Z 190,A -116.4878,B 1.0149,C 0.1893,E1 0.9445,E2 209.2803} C_DIS
LIN {X -78.4782,Y -108.5822,Z 190,A -114.7052,B 1.0145,C 0.1915,E1 0.9486,E2 207.4868} C_DIS
LIN {X -75.5511,Y -110.6391,Z 190,A -113.1737,B 1.0141,C 0.1934,E1 0.9522,E2 205.955} C_DIS
LIN {X -73.0575,Y -112.301,Z 190,A -111.7597,B 1.0139,C 0.1948,E1 0.9555,E2 204.5223} C_DIS
LIN {X -70.0505,Y -114.2008,Z 190,A -110.196,B 1.0136,C 0.1964,E1 0.9593,E2 202.9525} C_DIS
LIN {X -67.2373,Y -115.8795,Z 190,A -108.7315,B 1.0133,C 0.1978,E1 0.9629,E2 201.4789} C_DIS
LIN {X -64.3822,Y -117.49,Z 190,A -107.1314,B 1.0131,C 0.1989,E1 0.9669,E2 199.8509} C_DIS
LIN {X -61.6959,Y -118.9218,Z 190,A -105.8815,B 1.0128,C 0.2002,E1 0.97,E2 198.6079} C_DIS
LIN {X -58.7635,Y -120.3973,Z 190,A -104.4169,B 1.0126,C 0.2012,E1 0.9737,E2 197.1345} C_DIS
LIN {X -55.5284,Y -121.9243,Z 190,A -102.7983,B 1.0124,C 0.2023,E1 0.9779,E2 195.5032} C_DIS
LIN {X -52.6376,Y -123.1989,Z 190,A -101.4213,B 1.0122,C 0.2032,E1 0.9815,E2 194.1222} C_DIS
LIN {X -49.5,Y -124.4931,Z 190,A -99.8202,B 1.0121,C 0.2039,E1 0.9857,E2 192.4996} C_DIS
LIN {X -46.4414,Y -125.6659,Z 190,A -98.4893,B 1.0119,C 0.2048,E1 0.9892,E2 191.1782} C_DIS
LIN {X -43.3533,Y -126.7643,Z 190,A -97.0604,B 1.0118,C 0.2054,E1 0.9931,E2 189.745} C_DIS
LIN {X -40.4622,Y -127.7157,Z 190,A -95.695,B 1.0117,C 0.2058,E1 0.9968,E2 188.3702} C_DIS
LIN {X -37.0411,Y -128.7507,Z 190,A -94.1691,B 1.0116,C 0.2064,E1 1.0009,E2 186.8442} C_DIS
LIN {X -33.8713,Y -129.6209,Z 190,A -92.7451,B 1.0115,C 0.2068,E1 1.0048,E2 185.4172} C_DIS
LIN {X -30.3321,Y -130.4938,Z 190,A -91.2814,B 1.0114,C 0.2073,E1 1.0088,E2 183.9662} C_DIS
LIN {X -27.0992,Y -131.203,Z 190,A -89.8659,B 1.0114,C 0.2075,E1 1.0127,E2 182.5503} C_DIS
LIN {X -24.2525,Y -131.76,Z 190,A -88.4656,B 1.0114,C 0.2073,E1 1.0166,E2 181.1269} C_DIS
LIN {X -21.2803,Y -132.2732,Z 190,A -87.1101,B 1.0114,C 0.2071,E1 1.0205,E2 179.7617} C_DIS
LIN {X -17.8038,Y -132.7842,Z 190,A -85.7652,B 1.0114,C 0.2074,E1 1.0242,E2 178.4383} C_DIS
LIN {X -14.5012,Y -133.1849,Z 190,A -84.3534,B 1.0114,C 0.2074,E1 1.0281,E2 177.0274} C_DIS
LIN {X -11.5093,Y -133.4769,Z 190,A -83.0111,B 1.0114,C 0.2069,E1 1.0319,E2 175.6765} C_DIS
LIN {X -7.9286,Y -133.7375,Z 190,A -81.5099,B 1.0115,C 0.2066,E1 1.0361,E2 174.1794} C_DIS
LIN {X -4.0949,Y -133.9099,Z 190,A -80.0478,B 1.0115,C 0.2066,E1 1.0402,E2 172.7417} C_DIS
LIN {X -1.6592,Y -133.963,Z 190,A -78.804,B 1.0117,C 0.2056,E1 1.0438,E2 171.4689} C_DIS
LIN {X 0.9699,Y -133.9666,Z 190,A -77.9953,B 1.0117,C 0.206,E1 1.046,E2 170.704} C_DIS
Enddeposition()
LIN {X 0.9699,Y -133.9666,Z 190,A -77.9953,B 1.0117,C 0.206,E1 1.046,E2 170.704} C_DIS
Startdeposition()
$VEL.CP = VEL_PRINT
LIN {X -1.9148,Y -134.8577,Z 190,A -79.3594,B 1.0111,C 0.2074,E1 1.0417,E2 172.1133} C_DIS
LIN {X -4.9762,Y -134.7794,Z 190,A -80.9114,B 1.0108,C 0.2086,E1 1.0372,E2 173.7015} C_DIS
LIN {X -9.9873,Y -134.5007,Z 190,A -82.9616,B 1.0108,C 0.2089,E1 1.0315,E2 175.7412} C_DIS
LIN {X -14.41,Y -134.0988,Z 190,A -84.8267,B 1.0108,C 0.2092,E1 1.0262,E2 177.6041} C_DIS
LIN {X -17.6102,Y -133.7161,Z 190,A -86.2139,B 1.0107,C 0.2094,E1 1.0223,E2 178.9944} C_DIS
LIN {X -21.3243,Y -133.1761,Z 190,A -87.9698,B 1.0106,C 0.2098,E1 1.0173,E2 180.7738} C_DIS
LIN {X -25.2574,Y -132.4846,Z 190,A -89.5213,B 1.0106,C 0.2093,E1 1.0131,E2 182.3056} C_DIS
LIN {X -28.6429,Y -131.7942,Z 190,A -90.8891,B 1.0108,C 0.2089,E1 1.0093,E2 183.6599} C_DIS
LIN {X -31.6272,Y -131.1099,Z 190,A -92.3221,B 1.0108,C 0.2089,E1 1.0053,E2 185.112} C_DIS
LIN {X -35.5184,Y -130.112,Z 190,A -93.9697,B 1.0108,C 0.2083,E1 1.0009,E2 186.752} C_DIS
LIN {X -38.1936,Y -129.3499,Z 190,A -95.1926,B 1.011,C 0.208,E1 0.9975,E2 187.9811} C_DIS
LIN {X -41.691,Y -128.2668,Z 190,A -96.9259,B 1.011,C 0.2077,E1 0.9928,E2 189.7399} C_DIS
LIN {X -47.2954,Y -126.3059,Z 190,A -99.0409,B 1.0114,C 0.2056,E1 0.9873,E2 191.7982} C_DIS
LIN {X -49.5598,Y -125.4369,Z 190,A -100.4033,B 1.0114,C 0.2056,E1 0.9836,E2 193.2079} C_DIS
LIN {X -52.3059,Y -124.3151,Z 190,A -101.7536,B 1.0116,C 0.2049,E1 0.98,E2 194.571} C_DIS
LIN {X -56.2605,Y -122.5761,Z 190,A -103.7928,B 1.0118,C 0.2039,E1 0.9747,E2 196.6393} C_DIS
LIN {X -60.5366,Y -120.5232,Z 190,A -105.6899,B 1.0122,C 0.2021,E1 0.9699,E2 198.5204} C_DIS
LIN {X -63.0902,Y -119.2049,Z 190,A -106.943,B 1.0124,C 0.201,E1 0.9668,E2 199.7782} C_DIS
LIN {X -67.1781,Y -116.9522,Z 190,A -109.1331,B 1.0127,C 0.1993,E1 0.9613,E2 201.9977} C_DIS
LIN {X -70.4624,Y -115.0026,Z 190,A -110.8945,B 1.013,C 0.1978,E1 0.957,E2 203.7787} C_DIS
LIN {X -74.0893,Y -112.7002,Z 190,A -112.8028,B 1.0134,C 0.1957,E1 0.9525,E2 205.6989} C_DIS
LIN {X -77.4207,Y -110.4388,Z 190,A -114.5404,B 1.0138,C 0.1936,E1 0.9484,E2 207.4404} C_DIS
LIN {X -79.7582,Y -108.7621,Z 190,A -115.9702,B 1.0141,C 0.1923,E1 0.9451,E2 208.8991} C_DIS
LIN {X -83.2945,Y -106.0782,Z 190,A -117.9998,B 1.0145,C 0.1898,E1 0.9405,E2 210.9488} C_DIS
LIN {X -86.7358,Y -103.2833,Z 190,A -120.0074,B 1.015,C 0.1871,E1 0.9361,E2 212.9736} C_DIS
LIN {X -90.0829,Y -100.3775,Z 190,A -122.5885,B 1.0155,C 0.1846,E1 0.9305,E2 215.6508} C_DIS
LIN {X -93.5164,Y -97.1875,Z 190,A -124.8005,B 1.0161,C 0.1815,E1 0.9259,E2 217.893} C_DIS
LIN {X -96.9238,Y -93.7888,Z 190,A -126.6084,B 1.0167,C 0.1778,E1 0.9225,E2 219.6684} C_DIS
LIN {X -99.917,Y -90.5933,Z 190,A -128.5342,B 1.0173,C 0.1745,E1 0.9188,E2 221.603} C_DIS
LIN {X -102.8004,Y -87.3077,Z 190,A -130.5428,B 1.0179,C 0.171,E1 0.915,E2 223.6321} C_DIS
LIN {X -105.5164,Y -84.005,Z 190,A -132.5719,B 1.0184,C 0.1675,E1 0.9114,E2 225.69} C_DIS
LIN {X -108.1702,Y -80.5591,Z 190,A -134.5607,B 1.019,C 0.1638,E1 0.908,E2 227.6976} C_DIS
LIN {X -110.4659,Y -77.3823,Z 190,A -136.5543,B 1.0196,C 0.1604,E1 0.9047,E2 229.7354} C_DIS
LIN {X -113.0049,Y -73.624,Z 190,A -138.6914,B 1.0202,C 0.1562,E1 0.9013,E2 231.9005} C_DIS
LIN {X -115.0287,Y -70.4199,Z 190,A -140.4563,B 1.0208,C 0.1526,E1 0.8987,E2 233.6857} C_DIS
LIN {X -116.983,Y -67.1242,Z 190,A -142.1758,B 1.0213,C 0.1489,E1 0.8962,E2 235.4173} C_DIS
LIN {X -118.7211,Y -63.9991,Z 190,A -144.0192,B 1.0218,C 0.1453,E1 0.8937,E2 237.3036} C_DIS
LIN {X -120.2814,Y -61.0116,Z 190,A -145.5646,B 1.0223,C 0.1419,E1 0.8917,E2 238.8636} C_DIS
LIN {X -121.7755,Y -57.9721,Z 190,A -147.2183,B 1.0228,C 0.1384,E1 0.8896,E2 240.5455} C_DIS
LIN {X -123.2253,Y -54.8235,Z 190,A -148.9306,B 1.0233,C 0.1347,E1 0.8876,E2 242.2891} C_DIS
LIN {X -124.6181,Y -51.5805,Z 190,A -150.5706,B 1.0238,C 0.1309,E1 0.8858,E2 243.9472} C_DIS
LIN {X -125.7297,Y -48.8066,Z 190,A -152.5881,B 1.0242,C 0.1274,E1 0.8837,E2 246.0625} C_DIS
LIN {X -127.2215,Y -44.7786,Z 190,A -154.1041,B 1.0248,C 0.1229,E1 0.8823,E2 247.5374} C_DIS
LIN {X -128.6493,Y -40.4936,Z 190,A -156.336,B 1.0254,C 0.1177,E1 0.8803,E2 249.8095} C_DIS
LIN {X -129.5889,Y -37.3774,Z 190,A -158.2707,B 1.0258,C 0.1137,E1 0.8787,E2 251.8153} C_DIS
LIN {X -130.4415,Y -34.2829,Z 190,A -159.464,B 1.0262,C 0.1102,E1 0.8779,E2 252.986} C_DIS
LIN {X -131.2172,Y -31.182,Z 190,A -160.9868,B 1.0266,C 0.1064,E1 0.8769,E2 254.5296} C_DIS
LIN {X -131.8726,Y -28.2795,Z 190,A -162.5401,B 1.027,C 0.1028,E1 0.8759,E2 256.1196} C_DIS
LIN {X -132.6302,Y -24.4925,Z 190,A -164.5867,B 1.0275,C 0.0981,E1 0.8748,E2 258.2175} C_DIS
LIN {X -133.2978,Y -20.5382,Z 190,A -166.4647,B 1.0279,C 0.0933,E1 0.874,E2 260.1169} C_DIS
LIN {X -133.8038,Y -16.9412,Z 190,A -168.1686,B 1.0283,C 0.0889,E1 0.8733,E2 261.8406} C_DIS
LIN {X -134.1589,Y -13.8512,Z 190,A -169.6798,B 1.0286,C 0.0851,E1 0.8729,E2 263.3752} C_DIS
LIN {X -134.4262,Y -10.9494,Z 190,A -171.1653,B 1.0289,C 0.0814,E1 0.8725,E2 264.8914} C_DIS
LIN {X -134.6457,Y -7.8061,Z 190,A -172.7047,B 1.0292,C 0.0775,E1 0.8722,E2 266.4553} C_DIS
LIN {X -134.7862,Y -4.7996,Z 190,A -174.1701,B 1.0295,C 0.0738,E1 0.872,E2 267.9435} C_DIS
LIN {X -134.856,Y -2.0193,Z 190,A -175.5337,B 1.0297,C 0.0703,E1 0.872,E2 269.3291} C_DIS
LIN {X -134.8669,Y 1.1068,Z 190,A -177.2325,B 1.03,C 0.0663,E1 0.872,E2 271.0734} C_DIS
LIN {X -134.7714,Y 5.1806,Z 190,A -179.185,B 1.0303,C 0.0612,E1 0.8721,E2 273.0522} C_DIS
LIN {X -134.6087,Y 8.4052,Z 190,A 179.2654,B 1.0305,C 0.0573,E1 0.8724,E2 274.6231} C_DIS
LIN {X -134.364,Y 11.6856,Z 190,A 177.4842,B 1.0308,C 0.053,E1 0.8728,E2 276.4505} C_DIS
LIN {X -133.8702,Y 16.4036,Z 190,A 175.201,B 1.0311,C 0.0472,E1 0.8735,E2 278.7653} C_DIS
LIN {X -133.2786,Y 20.6624,Z 190,A 173.0798,B 1.0313,C 0.0419,E1 0.8744,E2 280.921} C_DIS
LIN {X -132.6533,Y 24.3636,Z 190,A 171.3406,B 1.0315,C 0.0374,E1 0.8752,E2 282.6769} C_DIS
LIN {X -131.9587,Y 27.8806,Z 190,A 168.7856,B 1.0316,C 0.0323,E1 0.8768,E2 285.3543} C_DIS
LIN {X -130.8231,Y 32.7954,Z 190,A 167.1087,B 1.0318,C 0.027,E1 0.8779,E2 286.9744} C_DIS
LIN {X -129.9464,Y 36.1115,Z 190,A 165.3187,B 1.0318,C 0.0228,E1 0.8792,E2 288.8031} C_DIS
LIN {X -128.7177,Y 40.2794,Z 190,A 163.2703,B 1.032,C 0.0178,E1 0.8809,E2 290.8744} C_DIS
LIN {X -127.7307,Y 43.3064,Z 190,A 161.7196,B 1.032,C 0.0141,E1 0.8822,E2 292.4476} C_DIS
LIN {X -126.0689,Y 47.928,Z 190,A 159.3161,B 1.032,C 0.0085,E1 0.8846,E2 294.887} C_DIS
LIN {X -124.9859,Y 50.6817,Z 190,A 157.8555,B 1.0321,C 0.0051,E1 0.8861,E2 296.3705} C_DIS
LIN {X -123.4088,Y 54.4132,Z 190,A 155.5567,B 1.0321,C 0.0005,E1 0.8888,E2 298.7351} C_DIS
LIN {X -122.0711,Y 57.3528,Z 190,A 154.3221,B 1.0321,C -0.0028,E1 0.8902,E2 299.953} C_DIS
LIN {X -120.6646,Y 60.2536,Z 190,A 152.6115,B 1.0321,C -0.0063,E1 0.8924,E2 301.7019} C_DIS
LIN {X -118.6485,Y 64.1342,Z 190,A 150.4977,B 1.0321,C -0.0109,E1 0.8952,E2 303.8437} C_DIS
LIN {X -116.6502,Y 67.7001,Z 190,A 148.5128,B 1.0321,C -0.015,E1 0.898,E2 305.8558} C_DIS
LIN {X -114.2099,Y 71.7408,Z 190,A 146.3764,B 1.0319,C -0.0196,E1 0.9011,E2 308.0057} C_DIS
LIN {X -111.9474,Y 75.223,Z 190,A 144.4248,B 1.0319,C -0.0235,E1 0.9042,E2 309.9774} C_DIS
LIN {X -109.9476,Y 78.1169,Z 190,A 142.5992,B 1.0318,C -0.0268,E1 0.9072,E2 311.8392} C_DIS
LIN {X -107.655,Y 81.2462,Z 190,A 140.8194,B 1.0317,C -0.0303,E1 0.9102,E2 313.6325} C_DIS
LIN {X -105.1094,Y 84.5139,Z 190,A 138.8876,B 1.0316,C -0.0338,E1 0.9136,E2 315.5824} C_DIS
Enddeposition()
END
